	COMPLETE:				
		robot.release(sectionID);
		
		aoiLoad.material := '';
		aoiLoad.execute := FALSE;
		
		loadCornerCardboardsEx := TRUE;
END_CASE
END_METHOD

METHOD loadCornerGuards : BOOL
VAR_INPUT
	pairIndex : INT;
END_VAR
VAR_OUTPUT
	error : BOOL;
END_VAR
VAR
	pair : REFERENCE TO PositionMaterials REF= materialsArr[pairIndex];
	errorLeft, errorRight : BOOL;
END_VAR
{warning disable C0371}

loadCornerGuards := 
	loadCornerGuardsEx(
		robot:= robotLeft, 
		aoiLoad:= aoiCornerGuardLeft, 
		loadStep:= loadStepLeft, 
		pairIndex:= pairIndex, 
		includeTopLeft:= TRUE, 
		includeTopRight:= FALSE, 
		includeBottomLeft:= TRUE, 
		includeBottomRight:= FALSE, 
		error=> errorLeft) 
	AND
	loadCornerGuardsEx(
		robot:= robotRight, 
		aoiLoad:= aoiCornerGuardRight, 
		loadStep:= loadStepRight, 
		pairIndex:= pairIndex, 
		includeTopLeft:= FALSE, 
		includeTopRight:= TRUE, 
		includeBottomLeft:= FALSE, 
		includeBottomRight:= TRUE, 
		error=> errorRight);
		
error := errorLeft OR errorRight;

(*
IF robotLeft.error OR robotRight.error THEN
	error := TRUE;
	RETURN;
	
ELSIF 
	(robotLeft.reservation <> sectionID AND_THEN NOT robotLeft.reserve(sectionID)) OR 
	(robotRight.reservation <> sectionID AND_THEN NOT robotRight.reserve(sectionID))
THEN //loading requires both robots be reserved together
	RETURN;
	
ELSIF //robots have wrong tool
	(robotLeft.tool <> sectionID AND_THEN NOT robotLeft.changeEOAT(targetTool := sectionID)) OR
	(robotRight.tool <> sectionID AND_THEN NOT robotRight.changeEOAT(targetTool := sectionID))
THEN
	RETURN;
	
END_IF

CASE loadStep OF
	0: //top and bottom
		IF aoiCornerGuardLeft.done AND aoiCornerGuardRight.done THEN
			aoiCornerGuardLeft.execute := aoiCornerGuardRight.execute := FALSE;
			aoiCornerGuardLeft.material := aoiCornerGuardRight.material := '';
			loadStep := 10;
			RETURN;
		END_IF
		
		aoiCornerGuardLeft.suctions := 0;
		aoiCornerGuardLeft.surfaceID := Surface.TOP;
		aoiCornerGuardLeft.material := pair.top;
		aoiCornerGuardLeft.numPads := 0;
		
		aoiCornerGuardRight.suctions := suctionBottom;
		aoiCornerGuardRight.surfaceID := Surface.BOTTOM;
		aoiCornerGuardRight.material := pair.bottom;
		aoiCornerGuardRight.numPads := 0;
		
		aoiCornerGuardLeft.execute := NOT aoiCornerGuardLeft.done AND NOT aoiCornerGuardLeft.busy;
		aoiCornerGuardRight.execute := NOT aoiCornerGuardRight.done AND NOT aoiCornerGuardRight.busy;
		
	10: //sides
		IF aoiCornerGuardLeft.done AND aoiCornerGuardRight.done THEN
			aoiCornerGuardLeft.execute := aoiCornerGuardRight.execute := FALSE;
			aoiCornerGuardLeft.material := aoiCornerGuardRight.material := '';
			loadStep := 10;
			RETURN;
		END_IF
		
		aoiCornerGuardLeft.suctions := 0;
		aoiCornerGuardLeft.surfaceID := Surface.LEFT;
		aoiCornerGuardLeft.material := pair.left;
		aoiCornerGuardLeft.numPads := 0;
		
		aoiCornerGuardRight.suctions := 0;
		aoiCornerGuardRight.surfaceID := Surface.RIGHT;
		aoiCornerGuardRight.material := pair.right;
		aoiCornerGuardRight.numPads := 0;
		
		aoiCornerGuardLeft.execute := NOT aoiCornerGuardLeft.done AND NOT aoiCornerGuardLeft.busy;
		aoiCornerGuardRight.execute := NOT aoiCornerGuardRight.done AND NOT aoiCornerGuardRight.busy;
		
	COMPLETE:
		loadStep := 0;
		loadCornerGuards := TRUE;
END_CASE

error := aoiCornerGuardLeft.error OR aoiCornerGuardRight.error;
*)
END_METHOD

METHOD loadCornerGuardsEx : BOOL
VAR_IN_OUT
	robot : RobotA22;
	aoiLoad : AOI_LoadCornerGuard;
	loadStep : INT;
END_VAR
VAR_INPUT
	pairIndex : INT;
	includeTopLeft, includeTopRight, includeBottomLeft, includeBottomRight : BOOL;
END_VAR
VAR_OUTPUT
	error : BOOL;
END_VAR
VAR
	pair : REFERENCE TO PositionMaterials REF= materialsArr[pairIndex];
END_VAR
{warning disable C0371}
IF robot.error THEN
	error := TRUE;
	RETURN;
ELSIF robot.reservation <> sectionID AND_THEN NOT robot.reserve(sectionID) THEN
	RETURN;
ELSIF robot.tool <> sectionID AND_THEN NOT robot.changeEOAT(targetTool := sectionID) THEN
	RETURN;
END_IF

error := aoiLoad.error;

CASE loadStep OF
	0:
		loadStep := Surface.BOTTOM_LEFT;
		
	Surface.BOTTOM_LEFT:
		IF NOT includeBottomLeft OR aoiLoad.donePulse THEN
			aoiLoad.execute := FALSE;
			aoiLoad.material := '';
			loadStep := Surface.BOTTOM_RIGHT;
			RETURN;
		END_IF
		
		aoiLoad.surfaceID := loadStep;
		aoiLoad.material := pair.bottomLeft;
		aoiLoad.suctions := suctionBottomLeft;
		aoiLoad.numPads := UPPER_BOUND(suctionBottomLeft, 1) - LOWER_BOUND(suctionBottomLeft, 1) + 1;
		
		aoiLoad.execute := NOT aoiLoad.busy;
		
	Surface.BOTTOM_RIGHT:
		IF NOT includeBottomRight OR aoiLoad.donePulse THEN
			aoiLoad.execute := FALSE;
			aoiLoad.material := '';
			loadStep := Surface.TOP_LEFT;
			RETURN;
		END_IF
		
		aoiLoad.surfaceID := loadStep;
		aoiLoad.material := pair.bottomRight;
		aoiLoad.suctions := suctionBottomRight;
		aoiLoad.numPads := UPPER_BOUND(suctionBottomRight, 1) - LOWER_BOUND(suctionBottomRight, 1) + 1;
		
		aoiLoad.execute := NOT aoiLoad.busy;
	
	Surface.TOP_LEFT:		
		IF NOT includeTopLeft OR aoiLoad.donePulse THEN
			aoiLoad.execute := FALSE;
			aoiLoad.material := '';
			loadStep := Surface.TOP_RIGHT;
			RETURN;
		END_IF
		
		aoiLoad.surfaceID := loadStep;
		aoiLoad.material := pair.top;
		aoiLoad.suctions := suctionTopLeft;
		aoiLoad.numPads := UPPER_BOUND(suctionTopLeft, 1) - LOWER_BOUND(suctionTopLeft, 1) + 1;
		
		aoiLoad.execute := NOT aoiLoad.busy;
		
	Surface.TOP_RIGHT:
		IF NOT includeTopRight OR aoiLoad.donePulse THEN
			aoiLoad.execute := FALSE;
			aoiLoad.material := '';
			loadStep := COMPLETE;
			RETURN;
		END_IF
		
		aoiLoad.surfaceID := loadStep;
		aoiLoad.material := pair.topRight;
		aoiLoad.suctions := suctionTopRight;
		aoiLoad.numPads := UPPER_BOUND(suctionTopRight, 1) - LOWER_BOUND(suctionTopRight, 1) + 1;
		
		aoiLoad.execute := NOT aoiLoad.busy;
		
	COMPLETE:				
		robot.release(sectionID);
		
		aoiLoad.material := '';
		aoiLoad.execute := FALSE;
		
		loadCornerGuardsEx := TRUE;
END_CASE
END_METHOD

METHOD PROTECTED loadFlatCardboards : BOOL
VAR_INPUT
	pairIndex : INT;
END_VAR
VAR_OUTPUT
	error : BOOL;
END_VAR
VAR
	pair : REFERENCE TO PositionMaterials REF= materialsArr[pairIndex];
	errorLeft, errorRight : BOOL;
END_VAR
{warning disable C0371}

loadFlatCardboards := 
	loadFlatCardboardsEx(
		robot:= robotLeft, 
		aoiLoad:= aoiFlatCardboardLeft, 
		loadStep:= loadStepLeft, 
		pairIndex:= pairIndex, 
		includeTop:= TRUE, 
		includeLeft:= FALSE, //left already loaded before
		includeRight:= FALSE, 
		includeBottom:= FALSE, 
		error=> errorLeft)
	AND
	loadFlatCardboardsEx(
		robot:= robotRight, 
		aoiLoad:= aoiFlatCardboardRight, 
		loadStep:= loadStepRight, 
		pairIndex:= pairIndex, 
		includeTop:= FALSE, 
		includeLeft:= FALSE, 
		includeRight:= FALSE, //right already loaded before
		includeBottom:= TRUE, 
		error=> errorRight);
		
error := errorLeft OR errorRight;

(*
IF robotLeft.error OR robotRight.error THEN
	error := TRUE;
	RETURN;
	
ELSIF 
	(robotLeft.reservation <> sectionID AND_THEN NOT robotLeft.reserve(sectionID)) OR 
	(robotRight.reservation <> sectionID AND_THEN NOT robotRight.reserve(sectionID))
THEN //loading requires both robots be reserved together
	RETURN;
	
ELSIF //robots have wrong tool
	(robotLeft.tool <> sectionID AND_THEN NOT robotLeft.changeEOAT(targetTool := sectionID)) OR
	(robotRight.tool <> sectionID AND_THEN NOT robotRight.changeEOAT(targetTool := sectionID))
THEN
	RETURN;
	
END_IF

CASE loadStep OF
	0: //top and bottom
		IF aoiFlatCardboardLeft.done AND aoiFlatCardboardRight.done THEN
			aoiFlatCardboardLeft.execute := aoiFlatCardboardRight.execute := FALSE;
			aoiFlatCardboardLeft.material := aoiFlatCardboardRight.material := '';
			loadStep := 10;
			RETURN;
		END_IF
		
		aoiFlatCardboardLeft.suctions := 0;
		aoiFlatCardboardLeft.surfaceID := Surface.TOP;
		aoiFlatCardboardLeft.material := pair.top;
		aoiFlatCardboardLeft.numPads := 0;
		
		aoiFlatCardboardRight.suctions := suctionBottom;
		aoiFlatCardboardRight.surfaceID := Surface.BOTTOM;
		aoiFlatCardboardRight.material := pair.bottom;
		aoiFlatCardboardRight.numPads := 0;
		
		aoiFlatCardboardLeft.execute := NOT aoiFlatCardboardLeft.done AND NOT aoiFlatCardboardLeft.busy;
		aoiFlatCardboardRight.execute := NOT aoiFlatCardboardRight.done AND NOT aoiFlatCardboardRight.busy;
		
	10: //sides
		IF aoiFlatCardboardLeft.done AND aoiFlatCardboardRight.done THEN
			aoiFlatCardboardLeft.execute := aoiFlatCardboardRight.execute := FALSE;
			aoiFlatCardboardLeft.material := aoiFlatCardboardRight.material := '';
			loadStep := 10;
			RETURN;
		END_IF
		
		aoiFlatCardboardLeft.suctions := 0;
		aoiFlatCardboardLeft.surfaceID := Surface.LEFT;
		aoiFlatCardboardLeft.material := pair.left;
		aoiFlatCardboardLeft.numPads := 0;
		
		aoiFlatCardboardRight.suctions := 0;
		aoiFlatCardboardRight.surfaceID := Surface.RIGHT;
		aoiFlatCardboardRight.material := pair.right;
		aoiFlatCardboardRight.numPads := 0;
		
		aoiFlatCardboardLeft.execute := NOT aoiFlatCardboardLeft.done AND NOT aoiFlatCardboardLeft.busy;
		aoiFlatCardboardRight.execute := NOT aoiFlatCardboardRight.done AND NOT aoiFlatCardboardRight.busy;
		
	COMPLETE:
		loadStepLeft := loadStepRight := 0;
		loadStep := 0;
		
		loadFlatCardboards := TRUE;
END_CASE

error := aoiFlatCardboardLeft.error OR aoiFlatCardboardRight.error;
*)
END_METHOD

METHOD loadFlatCardboardsEx : BOOL
VAR_IN_OUT
	robot : RobotA22;
	aoiLoad : AOI_LoadFlatCardboard;
	loadStep : INT;
END_VAR
VAR_INPUT
	pairIndex : INT;
	includeTop, includeLeft, includeRight, includeBottom : BOOL;
END_VAR
VAR_OUTPUT
	error : BOOL;
END_VAR
VAR
	pair : REFERENCE TO PositionMaterials REF= materialsArr[pairIndex];
END_VAR
IF robot.error THEN
	error := TRUE;
	RETURN;
ELSIF robot.reservation <> sectionID AND_THEN NOT robot.reserve(sectionID) THEN
	RETURN;
ELSIF robot.tool <> sectionID AND_THEN NOT robot.changeEOAT(targetTool := sectionID) THEN
	RETURN;
END_IF

error := aoiLoad.error;

CASE loadStep OF
	0:
		loadStep := Surface.TOP;
	
	Surface.TOP:	
		IF NOT includeTop OR aoiLoad.donePulse THEN
			aoiLoad.execute := FALSE;
			aoiLoad.material := '';
			loadStep := Surface.BOTTOM;
			RETURN;
		END_IF
		
		aoiLoad.surfaceID := Surface.TOP;
		aoiLoad.material := pair.top;
		aoiLoad.suctions := 0;
		aoiLoad.numPads := 0;
		
		aoiLoad.execute := NOT aoiLoad.busy;
		
	Surface.BOTTOM:
		IF NOT includeBottom OR aoiLoad.donePulse THEN
			aoiLoad.execute := FALSE;
			aoiLoad.material := '';
			loadStep := Surface.LEFT;
			RETURN;
		END_IF
		
		aoiLoad.surfaceID := Surface.BOTTOM;
		aoiLoad.material := pair.bottom;
		aoiLoad.suctions := suctionBottom;
		aoiLoad.numPads := UPPER_BOUND(suctionBottom, 1) - LOWER_BOUND(suctionBottom, 1) + 1;
		
		aoiLoad.execute := NOT aoiLoad.busy;
		
	Surface.LEFT:
		IF NOT includeLeft OR aoiLoad.donePulse THEN
			aoiLoad.execute := FALSE;
			aoiLoad.material := '';
			loadStep := Surface.RIGHT;
			RETURN;
		END_IF
		
		aoiLoad.surfaceID := Surface.LEFT;
		aoiLoad.material := pair.left;
		aoiLoad.suctions := 0;
		aoiLoad.numPads := 0;
		
		aoiLoad.execute := NOT aoiLoad.busy;
		
	Surface.RIGHT:
		IF NOT includeRight OR aoiLoad.donePulse THEN
			aoiLoad.execute := FALSE;
			aoiLoad.material := '';
			loadStep := COMPLETE;
			RETURN;
		END_IF
		
		aoiLoad.surfaceID := Surface.RIGHT;
		aoiLoad.material := pair.right;
		aoiLoad.suctions := 0;
		aoiLoad.numPads := 0;
		
		aoiLoad.execute := NOT aoiLoad.busy;
		
	COMPLETE:				
		robot.release(sectionID);
		
		aoiLoad.material := '';
		aoiLoad.execute := FALSE;
		
		loadFlatCardboardsEx := TRUE;
END_CASE
END_METHOD

METHOD PROTECTED maintenance : BOOL
VAR_INPUT
END_VAR
{warning disable C0371}
IF robotLeft.Done THEN
	robotLeft.clearCommand();
END_IF

IF robotRight.Done THEN
	robotRight.clearCommand();
END_IF
END_METHOD

METHOD PROTECTED manual : BOOL
VAR_INPUT
END_VAR
END_METHOD

METHOD PROTECTED process : BOOL
VAR_INPUT
	auto : BOOL;
END_VAR
VAR_OUTPUT
	error : BOOL;
END_VAR
VAR
	currentPair : REFERENCE TO PositionMaterials REF= materialsArr[iPair];
END_VAR
{warning disable C0371}

IF iPair >= CONSTS.maxPairs THEN
	process := TRUE;
	RETURN;
ELSIF NOT PositionIsValid(pair := currentPair) THEN
	iPair := iPair + 1;
	RETURN;
END_IF
(*
corrected sequence:
	load sides
	load corners
	load bottom
	load top
*)

CASE step OF
	IDLE:
		IF execute THEN
			execute := FALSE;
			step := LOAD_SIDES_CORNERS;
		END_IF
	
	LOAD_SIDES_CORNERS:
		IF
			(auto AND done) OR
			(NOT auto AND execute)
		THEN
			aoiCornerCardboardLeft.reset();
			aoiCornerCardboardRight.reset();
			
			aoiCornerGuardLeft.reset();
			aoiCornerGuardRight.reset();
			
			aoiFlatCardboardLeft.reset();
			aoiFlatCardboardRight.reset();
			
			step := LOAD_TOP_BOTTOM;
			RETURN;
		END_IF
		
		IF NOT done THEN
			done := load(pairIndex := iPair);
		END_IF
		
	LOAD_TOP_BOTTOM:
		IF
			(auto AND done) OR
			(NOT auto AND execute)
		THEN
			aoiCornerCardboardLeft.reset();
			aoiCornerCardboardRight.reset();
			
			aoiCornerGuardLeft.reset();
			aoiCornerGuardRight.reset();
			
			aoiFlatCardboardLeft.reset();
			aoiFlatCardboardRight.reset();
			
			step := PUSH;
			RETURN;
		END_IF
		
		IF NOT done THEN
			done := loadFlatCardboards(pairIndex := iPair);
		END_IF
		
	PUSH:
		IF
			(auto AND latchLeft AND latchRight AND pistonBottom.extended) OR
			(NOT auto AND execute)
		THEN
			step := TARGET_WRAP_POSITION;
			RETURN;
		END_IF
		
		insertionLeft.align(demoHeight+5);
		insertionRight.align(demoHeight+5);
		
		IF //align slider to 5mm gap above bundle height
			insertionLeft.sliderPos <> demoHeight+5 OR
			insertionRight.sliderPos <> demoHeight+5
		THEN
			RETURN;
		END_IF
		
		IF NOT latchLeft THEN
			latchLeft := insertionLeft.contact;
			insertionLeft.press();
		END_IF
		
		IF NOT latchRight THEN
			latchRight := insertionRight.contact;
			insertionRight.press();
		END_IF
		
		pistonBottom.extend();
		
	TARGET_WRAP_POSITION:		
		IF iWrap >= wrapPoints THEN
			step := COMPLETE;
			RETURN;
		END_IF
		
		IF materialsArr[iPair].position = materialsArr[iPair + 1].position THEN //if this and the next pair were loaded together
			masterLength := TO_INT( MAX( GetPairMasterLength(materialsArr[iPair]), GetPairMasterLength(materialsArr[iPair + 1]) ) );
			wrapPoints := MAX( materialsArr[iPair].wrapPoints, materialsArr[iPair + 1].wrapPoints );
			wrapRotations := MAX( materialsArr[iPair].wrapRotations, materialsArr[iPair + 1].wrapRotations );
		ELSE
			masterLength := TO_INT( GetPairMasterLength(materialsArr[iPair]) );
			wrapPoints := materialsArr[iPair].wrapPoints;
			wrapRotations := materialsArr[iPair].wrapRotations;
		END_IF
		
		(*
		directionCheckAndSet(
			wrapConveyorPos,
			(currentPair.position - masterLength/2) + (masterLength/(currentPair.wrapPoints + 1) * (iWrap + 1)));
		*)
		step := WRAP_AND_RELEASE;
		
	WRAP_AND_RELEASE:
		releaseDelayTimer(IN:= , PT:= releaseDelay, Q=> , ET=> );
		
		IF wrapper.ready THEN
			wrapper.wrap(wrapRotations);
			releaseDelayTimer.IN := TRUE;
		END_IF
		
		IF releaseDelayTimer.Q THEN
			SetSuctions(suctions := suctionTopLeft, state := FALSE);
			SetSuctions(suctions := suctionTopRight, state := FALSE);
			SetSuctions(suctions := suctionBottomLeft, state := FALSE);
			SetSuctions(suctions := suctionBottomRight, state := FALSE);
			
			insertionLeft.toHome();
			insertionRight.toHome();
			pistonBottom.retract();
		END_IF
		
		IF wrapper.done AND insertionLeft.home AND insertionRight.home AND pistonBottom.retracted THEN
			releaseDelayTimer.IN := FALSE;
			step := WRAP_AND_RELEASE;
		END_IF
	
	COMPLETE:
		iPair := iPair + 1;
		iWrap := wrapPoints := wrapRotations := 0;
		step := IDLE;
		
END_CASE
END_METHOD

METHOD PROTECTED ps_AbortCondition : BOOL
VAR_INPUT
END_VAR
{warning disable C0371}
ps_AbortCondition :=
	insertionLeft.error OR 
	insertionRight.error OR 
	robotLeft.error OR 
	robotRight.error OR
	wrapper.error;
END_METHOD

METHOD PROTECTED ps_Aborted : BOOL
VAR_INPUT
END_VAR
ps_Aborted := TRUE;
END_METHOD

METHOD PROTECTED ps_Aborting : BOOL
VAR_INPUT
END_VAR
{warning disable C0371}
insertionLeft.stop();
insertionRight.stop();
pistonBottom.stop();

aoiFlatCardboardLeft.reset();
aoiFlatCardboardRight.reset();

aoiCornerCardboardLeft.reset();
aoiCornerCardboardRight.reset();

aoiCornerGuardLeft.reset();
aoiCornerGuardRight.reset();

robotLeft.clearCommand();
robotRight.clearCommand();

//stop conveyors

ps_Aborting :=
	NOT insertionLeft.active AND
	NOT insertionRight.active AND
	NOT pistonBottom.busy AND
	NOT robotLeft.Busy AND
	NOT robotRight.Busy;
END_METHOD

METHOD PROTECTED ps_Clearing : BOOL
VAR_INPUT
END_VAR
{warning disable C0371}
insertionLeft.reset();
insertionRight.reset();

ps_Clearing := 
	NOT insertionLeft.error AND
	NOT insertionRight.error AND
	NOT wrapper.error AND
	NOT robotLeft.error AND
	NOT robotRight.error;
END_METHOD

METHOD PROTECTED ps_Complete : BOOL
VAR_INPUT
END_VAR
ps_Complete := TRUE;
END_METHOD

METHOD PROTECTED ps_Completing : BOOL
VAR_INPUT
END_VAR
ps_Completing := NOT occupied;
END_METHOD

METHOD PROTECTED ps_Execute : BOOL
VAR_INPUT
END_VAR
VAR_OUTPUT
	error : BOOL;
END_VAR
CASE pmlMode OF
	0: //invalid mode
	ePMLCustomUnitMode_Production:		ps_Execute := process(auto := TRUE, error => error);
	ePMLCustomUnitMode_Maintenance:		ps_Execute := maintenance();
	ePMLCustomUnitMode_Manual:			ps_Execute := manual();
	ePMLCustomUnitMode_SemiAuto:		ps_Execute := process(auto := FALSE, error => error);
END_CASE
END_METHOD

METHOD PROTECTED ps_Held : BOOL
VAR_INPUT
END_VAR
ps_Held := NOT hold;
END_METHOD

METHOD PROTECTED ps_HoldCondition : BOOL
VAR_INPUT
END_VAR
END_METHOD

METHOD PROTECTED ps_Holding : BOOL
VAR_INPUT
END_VAR
{warning disable C0371}
insertionLeft.stop();
insertionRight.stop();
pistonBottom.stop();
//set robot to pause

ps_Holding :=
	NOT insertionLeft.active AND
	NOT insertionRight.active;
END_METHOD

METHOD PROTECTED ps_Idle : BOOL
VAR_INPUT
END_VAR
ps_Idle := execute;
execute := FALSE;
END_METHOD

METHOD PROTECTED ps_Resetting : BOOL
VAR_INPUT
END_VAR
{warning disable C0371}
insertionLeft.reset();
insertionRight.reset();

ps_Resetting := 
	reset AND
	NOT insertionLeft.error AND
	NOT insertionRight.error AND
	NOT wrapper.error AND
	NOT robotLeft.error AND
	NOT robotRight.error;
END_METHOD

METHOD PROTECTED ps_Starting : BOOL
VAR_INPUT
END_VAR
{warning disable C0371}
robotLeft.clearCommand();
robotRight.clearCommand();

insertionLeft.homingSequence();
insertionRight.homingSequence();
pistonBottom.retract();

ps_Starting := 
	insertionLeft.screw.HomeSet AND 
	insertionRight.screw.HomeSet AND 
	pistonBottom.retracted;
END_METHOD

METHOD PROTECTED ps_StopCondition : BOOL
VAR_INPUT
END_VAR
ps_StopCondition := 
	stop;
END_METHOD

METHOD PROTECTED ps_Stopped : BOOL
VAR_INPUT
END_VAR
ps_Stopped := TRUE;
END_METHOD

METHOD PROTECTED ps_Stopping : BOOL
VAR_INPUT
END_VAR
{warning disable C0371}
insertionLeft.stop();
insertionRight.stop();
pistonBottom.stop();

aoiFlatCardboardLeft.reset();
aoiFlatCardboardRight.reset();

aoiCornerCardboardLeft.reset();
aoiCornerCardboardRight.reset();

aoiCornerGuardLeft.reset();
aoiCornerGuardRight.reset();

robotLeft.clearCommand();
robotRight.clearCommand();

wrapper.bEnable := FALSE;

//stop conveyors

ps_Stopping :=
	//NOT insertionLeft.active AND
	NOT insertionRight.active AND
	NOT pistonBottom.busy AND
	NOT robotLeft.Busy AND
	NOT robotRight.Busy AND
	NOT wrapper.busy;
END_METHOD

METHOD PROTECTED ps_SuspendCondition : BOOL
VAR_INPUT
END_VAR
END_METHOD

METHOD PROTECTED ps_Suspended : BOOL
VAR_INPUT
END_VAR
ps_Suspended := NOT ps_SuspendCondition();
END_METHOD

METHOD PROTECTED ps_Suspending : BOOL
VAR_INPUT
END_VAR
ps_Suspending := TRUE;
END_METHOD

METHOD PROTECTED ps_Unholding : BOOL
VAR_INPUT
END_VAR
ps_Unholding := TRUE;
END_METHOD

METHOD PROTECTED ps_Unsuspending : BOOL
VAR_INPUT
END_VAR
ps_Unsuspending := TRUE;
END_METHOD

METHOD PROTECTED FINAL runSectionTasks : BOOL
VAR_INPUT
	auto : BOOL;
END_VAR
VAR_OUTPUT
	error : BOOL;
END_VAR
SUPER^.runSectionTasks(auto := auto, error => error);

CASE status OF
	SectionTask.IDLE:
		RETURN;
	
	SectionTask.ALIGNING:
		IF NOT recipesCombined THEN
			combine(
				currentBundle.cardboard, 
				currentBundle.cornerGuard, 
				materialsArr, 
				currentBundle.cardboard_over_cornerGuard);
				
			recipesCombined := TRUE;
		END_IF
		
	SectionTask.ACTIVE:
		recipesCombined := FALSE;
		
	SectionTask.CLEARING:
		//
		
	SectionTask.COMPLETE:	
		//
		
	-100:
		RETURN;
		
END_CASE
END_METHOD

METHOD PROTECTED setOrder : BOOL
VAR_IN_OUT
	innerArray : ARRAY[*] OF PositionMaterials;
	outerArray : ARRAY[*] OF PositionMaterials;
	
	combined : ARRAY[*] OF PositionMaterials;
	
	i_inner : INT;
	i_outer : INT;
	i_combined : INT;
END_VAR
VAR	
	outerMaterialLength : LREAL;
	innerMaterialLength : LREAL;
END_VAR
//if inner material is in front of outer material, inner material goes first
IF innerArray[i_inner].position <= outerArray[i_outer].position THEN

	combined[i_combined] := innerArray[i_inner];
	i_inner := i_inner + 1; //check next cardboard during next iteration
	
	setOrder := TRUE;
	RETURN;
END_IF
	
outerMaterialLength := GetPairMasterLength(outerArray[i_outer]);
innerMaterialLength := GetPairMasterLength(innerArray[i_inner]);

//if current inner material is too close to current outer material, place inner material first
//compare inner materials' front with outer material's back
IF (innerArray[i_inner].position - innerMaterialLength/2) < (outerArray[i_outer].position + outerMaterialLength/2) THEN
	combined[i_combined] := innerArray[i_inner];
	i_inner := i_inner + 1;
ELSE //otherwise, outer material can go
	combined[i_combined] := outerArray[i_outer];
	i_outer := i_outer + 1;
END_IF

setOrder := TRUE;
END_METHOD

METHOD PROTECTED unload : BOOL
VAR_INPUT
END_VAR
END_METHOD

END_FUNCTION_BLOCK

// ---- Sections/Abstract/SectionEx.TcPOU
FUNCTION_BLOCK ABSTRACT SectionEx
VAR_INPUT
	enable : BOOL;
	sectionID : SectionEnum;
END_VAR
VAR_IN_OUT
	bundlesQueue : ARRAY[*] OF Bundle;
	bundlesBypass : ARRAY[*] OF BOOL; //if true, then bypass current bundle
	
	conveyorsArr : ARRAY[*] OF POINTER TO ConveyorSC;
	//in addition to the conveyos array, each section must receive references to the origial conveyors the array elements point to
END_VAR
VAR_OUTPUT
	bundleOut : Bundle; //assigned if there is a bundle to target
	bypass : BOOL; //assigned once the bundle head passes the section (status >= ACTIVE)
END_VAR
VAR_OUTPUT //PackML states + controls
	run : BOOL;
	stop : BOOL;
	execute : BOOL;
	hold : BOOL;
	reset : BOOL;
	
	ready : BOOL;
	busy : BOOL;
	done : BOOL;
	error : BOOL;
	
	pmlModeString : STRING;
	pmlStateString : STRING;
	
	pmlState : E_PMLState;
	pmlMode : E_PMLCustomUnitMode;
	
	iBundle : INT(0..Consts.maxQueue);
	iPair : INT(0..Consts.maxPairs);
END_VAR
VAR //PackML types
	pmlCommand : E_PMLCommand;
	pmlModeRequest : E_PMLCustomUnitMode := ePMLCustomUnitMode_Production;
	
	pmlStateMachine : PML_StateMachine;
	pmlModeManager : PML_UnitModeManager;
	pmlSemiAutoConfig : PML_UnitModeConfig;
END_VAR
VAR
	currentBundle : REFERENCE TO Bundle;
	currentBypass : REFERENCE TO BOOL;
	
	loaded : BOOL;
	loadedMaterials : ARRAY[Surface.TOP..Surface.BOTTOM_RIGHT] OF STRING;
	
	entryRefPos : (*REFERENCE TO*) REAL;
	exitRefPos : (*REFERENCE TO*) REAL;
	
	requestedConveyorMode : ConveyorMode;
	
	nextSection : POINTER TO SectionEx;
	prevSection : POINTER TO SectionEx;
	
	occupied : BOOL; //may need to move this to Hardware GVL since this is a sensor
	
	status : SectionTask; //section status
END_VAR
VAR_STAT CONSTANT
	INCLUSIVE : INT := 0;
	EXCLUSIVE : INT := 1;
	COMPLETE : INT := 1030;
	
	suctionReleaseDelay : TIME := T#1000MS;
END_VAR

currentBundle REF= bundlesQueue[iBundle];
currentBypass REF= bundlesBypass[iBundle];
bypass := currentBypass;

ready := status = 0;
busy := status > 0;
done := done;
error := error;

blocks();

configPmlModes();
runPmlStates();

METHOD PROTECTED blocks : BOOL
pmlModeManager(
	bExecute:= NOT pmlModeManager.bExecute, 
	eModeCommand:= pmlModeRequest, 
	eState:= pmlState, 
	eModeStatus=> pmlMode, 
	sModeStatus=> pmlModeString, 
	bDone=> , 
	bError=> , 
	nErrorId=> );

pmlStateMachine(
	eMode:= pmlMode, 
	eCommand:= pmlCommand, 
	stSubUnitInfoRef:= , 
	stOptions:= , 
	eState=> pmlState, 
	sState=> pmlStateString, 
	bError=> , 
	nErrorID=> );
END_METHOD

METHOD PROTECTED configPmlModes : BOOL
pmlSemiAutoConfig(
	eMode:= 4, 
	sName:= 'SemiAuto', 
	bDisableClearing:= FALSE, 
	bDisableStarting:= FALSE, 
	bDisableSuspended:= FALSE, 
	bDisableStopping:= FALSE, 
	bDisableAborting:= FALSE, 
	bDisableHolding:= FALSE, 
	bDisableHeld:= FALSE, 
	bDisableUnholding:= FALSE, 
	bDisableSuspending:= FALSE, 
	bDisableUnsuspending:= FALSE, 
	bDisableResetting:= FALSE, 
	bDisableIdle:= FALSE, 
	bDisableCompleting:= FALSE, 
	bDisableComplete:= FALSE, 
	bEnableUnitModeChangeStopped:= TRUE, 
	bEnableUnitModeChangeIdle:= TRUE, 
	bEnableUnitModeChangeSuspended:= FALSE, 
	bEnableUnitModeChangeExecute:= FALSE, 
	bEnableUnitModeChangeAborted:= TRUE, 
	bEnableUnitModeChangeHeld:= FALSE, 
	bEnableUnitModeChangeComplete:= FALSE, 
	bError=> , 
	nErrorId=> );
END_METHOD

METHOD connectTo : BOOL
VAR_INPUT
	connectedSection : POINTER TO SectionEx;
END_VAR
nextSection := connectedSection;

IF connectedSection <> 0 THEN
	connectedSection^.prevSection := THIS;
END_IF
END_METHOD

METHOD PROTECTED directionCheckAndSet : BOOL
VAR_INPUT
	conveyorRef : REAL;
	target : REAL;
END_VAR
//returns true conveyorRef is in range of target
IF InRange(conveyorRef - CONSTS.precisionTolerance, conveyorRef + CONSTS.precisionTolerance, target, EXCLUSIVE) THEN
	directionCheckAndSet := TRUE;
	
ELSIF conveyorRef > target THEN
	pConveyorMode := ConveyorMode.BACKWARD;
	
ELSIF conveyorRef < target THEN
	pConveyorMode := ConveyorMode.FORWARD;
	
END_IF
END_METHOD

METHOD PROTECTED ABSTRACT load : BOOL
VAR_INPUT
	pairIndex : INT;
END_VAR
VAR_OUTPUT
	error : BOOL;
END_VAR
(*
loading takes place while the section is NOT active
materials are loaded for the next incoming bundle, not the current bundle - may differ for each section
*)
END_METHOD

METHOD PROTECTED ABSTRACT maintenance : BOOL
VAR_INPUT
END_VAR
END_METHOD

METHOD PROTECTED ABSTRACT manual : BOOL
VAR_INPUT
END_VAR
END_METHOD

PROPERTY PROTECTED pConveyorMode : ConveyorMode
GET
pConveyorMode := requestedConveyorMode;
END_GET
SET
VAR
	i : DINT;
END_VAR
requestedConveyorMode := pConveyorMode;

FOR i:=LOWER_BOUND(conveyorsArr, 1) TO UPPER_BOUND(conveyorsArr, 1) BY 1 DO
	
	CASE status OF
		SectionTask.ALIGNING, -100:
			//all conveyors requested to same mode
			conveyorsArr[i]^.setRequest(requestedConveyorMode);
			
		SectionTask.ACTIVE, SectionTask.CLEARING:
			//once previous bundle catches up, the conveyor that bundle sits on must be linked to this section
			//a conveyor control module will handle linking
			
			IF conveyorsArr[i]^.IsOccupied THEN //follow this section's request
				conveyorsArr[i]^.setRequest(requestedConveyorMode);
				
			ELSE //catch up succeeding bundle (FOLLOW PREVIOUS SECTION)
				IF prevSection <> 0 THEN
					conveyorsArr[i]^.setRequest( prevSection^.pConveyorMode );
				END_IF
			END_IF
	END_CASE	
	
END_FOR
END_SET
END_PROPERTY

METHOD PROTECTED ABSTRACT process : BOOL
VAR_INPUT
	auto : BOOL;
END_VAR
VAR_OUTPUT
	error : BOOL;
END_VAR
(*
this method is implemented by each section according to their material packaging steps
*)
END_METHOD

METHOD PROTECTED ABSTRACT ps_AbortCondition : BOOL
VAR_INPUT
END_VAR
END_METHOD

METHOD PROTECTED ABSTRACT ps_Aborted : BOOL
VAR_INPUT
END_VAR
END_METHOD

METHOD PROTECTED ABSTRACT ps_Aborting : BOOL
VAR_INPUT
END_VAR
END_METHOD

METHOD PROTECTED ABSTRACT ps_Clearing : BOOL
VAR_INPUT
END_VAR
END_METHOD

METHOD PROTECTED ABSTRACT ps_Complete : BOOL
VAR_INPUT
END_VAR
END_METHOD

METHOD PROTECTED ABSTRACT ps_Completing : BOOL
VAR_INPUT
END_VAR
END_METHOD

METHOD PROTECTED ps_Execute : BOOL
VAR_INPUT
END_VAR
VAR_OUTPUT
	error : BOOL;
END_VAR
CASE pmlMode OF
	0: //invalid mode
	ePMLCustomUnitMode_Production:		ps_Execute := runSectionTasks(auto := TRUE);
	ePMLCustomUnitMode_Maintenance:		ps_Execute := maintenance();
	ePMLCustomUnitMode_Manual:			ps_Execute := manual();
	ePMLCustomUnitMode_SemiAuto:		ps_Execute := runSectionTasks(auto := FALSE);
END_CASE
END_METHOD

METHOD PROTECTED ABSTRACT ps_Held : BOOL
VAR_INPUT
END_VAR
END_METHOD

METHOD PROTECTED ABSTRACT ps_HoldCondition : BOOL
VAR_INPUT
END_VAR
END_METHOD

METHOD PROTECTED ABSTRACT ps_Holding : BOOL
VAR_INPUT
END_VAR
END_METHOD

METHOD PROTECTED (*ABSTRACT*) ps_Idle : BOOL
VAR_INPUT
END_VAR
ps_Idle := run OR execute; (*start section input*)

IF execute THEN
	run := TRUE;
END_IF
END_METHOD

METHOD PROTECTED ABSTRACT ps_Resetting : BOOL
VAR_INPUT
END_VAR
END_METHOD

METHOD PROTECTED ABSTRACT ps_Starting : BOOL
VAR_INPUT
END_VAR
END_METHOD

METHOD PROTECTED ABSTRACT ps_StopCondition : BOOL
VAR_INPUT
END_VAR
END_METHOD

METHOD PROTECTED ABSTRACT ps_Stopped : BOOL
VAR_INPUT
END_VAR
END_METHOD

METHOD PROTECTED ABSTRACT ps_Stopping : BOOL
VAR_INPUT
END_VAR
END_METHOD

METHOD PROTECTED ABSTRACT ps_SuspendCondition : BOOL
VAR_INPUT
END_VAR
END_METHOD

METHOD PROTECTED ABSTRACT ps_Suspended : BOOL
VAR_INPUT
END_VAR
END_METHOD

METHOD PROTECTED ABSTRACT ps_Suspending : BOOL
VAR_INPUT
END_VAR
END_METHOD

METHOD PROTECTED ABSTRACT ps_Unholding : BOOL
VAR_INPUT
END_VAR
END_METHOD

METHOD PROTECTED ABSTRACT ps_Unsuspending : BOOL
VAR_INPUT
END_VAR
END_METHOD

PROPERTY PROTECTED pStatus : SectionTask
GET
pStatus := status;
END_GET
SET
status := pStatus;
END_SET
END_PROPERTY

METHOD PROTECTED runPmlStates : BOOL
(*
PackML
	state machine for packaging applications - see Tc3_PackML_V2 library on InfoSys
	
	final states - wait for an input or condition and command to new state
	intermediate states - complete a task and call pmlStateMachine.M_StateComplete() to advance to next state
	
the following states currently use the same logic (albeit in different methods), implementation may change later
	ps_Stopping() and ps_Aborting()
	ps_Resetting() and ps_Clearing()
	
STOP - controlled stop **with intent to shutdown or vacate for extended time** induced by operator/HMI - otherwise use HOLD
ABORT - emergency stop due to machine errors


HOLD - minor local issues
SUSPEND - external issues

EXECUTE - major control logic
	different modes may require different tasks
	create methods as required for different modes, then call the correct method in ps_Completing()
	can be commanded to STOP, ABORT, HOLD, or SUSPEND at any point
COMPLETING - process complete, move product out of system and finish transition to COMPLETED

the implementation below can be copied to all POUs that use a PackML state machine
the individual ps_< > methods need to be implemented for the specific application
*)


IF ps_AbortCondition() THEN //abort condition
	pmlCommand := ePMLCommand_Abort;
ELSIF ps_StopCondition() THEN //stop condition
	pmlCommand := ePMLCommand_Stop;
END_IF

CASE pmlState OF
	0 (*ePMLState_Undefined*): //default state on startup
		pmlCommand := ePMLCommand_Stop;
		
	ePMLState_Stopping:
		IF ps_Stopping() THEN
			pmlStateMachine.M_StateComplete();
		END_IF
		
	ePMLState_Stopped:
		IF ps_Stopped() THEN
			pmlCommand := ePMLCommand_Reset;
		END_IF
	
    ePMLState_Resetting:
		IF ps_Resetting() THEN
			pmlStateMachine.M_StateComplete();
		END_IF
		
	ePMLState_Idle:
		IF ps_Idle() THEN
			pmlCommand := ePMLCommand_Start;
		END_IF		
	
	ePMLState_Starting:
		IF ps_Starting() THEN
			pmlStateMachine.M_StateComplete();
		END_IF
	
	ePMLState_Execute: //check the conditions in order of their priority, currently HOLD has the highest priority
		IF ps_HoldCondition() THEN
			pmlCommand := ePMLCommand_Hold;
			
		ELSIF ps_SuspendCondition() THEN
			pmlCommand := ePMLCommand_Suspend;			
		
		ELSIF ps_Execute(error => error) THEN //ps_Execute.error => THIS^.error
			pmlStateMachine.M_StateComplete();
			pmlCommand := ePMLCommand_Complete;
		END_IF
		
	ePMLState_Completing:
		IF ps_Completing() THEN
			pmlStateMachine.M_StateComplete();
		END_IF
	
	ePMLState_Complete:
		IF ps_Complete() THEN
			pmlCommand := ePMLCommand_Reset;
		END_IF
	
	ePMLState_Holding:
		IF ps_Holding() THEN
			pmlStateMachine.M_StateComplete();
		END_IF
	
	ePMLState_Held:
		IF NOT hold THEN
			pmlCommand := ePMLCommand_Unhold;
		END_IF
	
	ePMLState_Unholding:
		IF ps_Unholding() THEN
			pmlStateMachine.M_StateComplete(); //release all pause commands and IO
		END_IF
		
	ePMLState_Suspending: //based on next section conditions
		IF ps_Suspending() THEN
			pmlStateMachine.M_StateComplete();
		END_IF
		
	ePMLState_Suspended: //based on next section conditions
		IF ps_Suspended() THEN
			pmlCommand := ePMLCommand_Unsuspend;
		END_IF
	
	ePMLState_Unsuspending: //based on next section conditions
		IF ps_Unsuspending() THEN
			pmlStateMachine.M_StateComplete();
		END_IF
	
	ePMLState_Aborting:
		IF ps_Aborting() THEN
			pmlStateMachine.M_StateComplete();
		END_IF
	
	ePMLState_Aborted:
		IF ps_Aborted() THEN
			pmlCommand := ePMLCommand_Clear;
		END_IF
	
	ePMLState_Clearing:
		IF ps_Clearing() THEN
			pmlStateMachine.M_StateComplete();
		END_IF
	
END_CASE
END_METHOD

METHOD PROTECTED runSectionTasks : BOOL
VAR_INPUT
	auto : BOOL;
END_VAR
VAR_OUTPUT
	error : BOOL;
END_VAR
CASE status OF
	SectionTask.IDLE:
		IF BundleIsValid(currentBundle) THEN			
			status := SectionTask.ALIGNING;
			done := FALSE;
		END_IF
	
	SectionTask.ALIGNING:		
		pConveyorMode := ConveyorMode.FORWARD;
		
		IF 
			occupied AND
			nextSection <> 0 AND
			nextSection^.pConveyorMode = ConveyorMode.BACKWARD
		THEN //section occupied by next section backing up into this section
			status := -100;
			
		ELSIF occupied THEN //section occupied by correct bundle
			//stop and zero the conveyors
			IF NOT auto OR_ELSE execute THEN
				status := SectionTask.ACTIVE;
			END_IF
		END_IF
		
	SectionTask.ACTIVE:
		bundleOut := currentBundle;
		
		IF NOT enable THEN
			iPair := 0;
			status := SectionTask.CLEARING;
			
		ELSIF currentBypass (*AND_THEN discharge()*) THEN //bundle failed in previous section, discharge this section's materials
			IF unload() THEN
				iPair := 0;
				status := SectionTask.CLEARING;
			END_IF
			
		ELSIF process(auto := auto, error => error) THEN //bundle recipe completed normally
			IF NOT auto OR_ELSE execute THEN
				iPair := 0;
				status := SectionTask.CLEARING;
			END_IF			
		END_IF
		
	SectionTask.CLEARING:
		bundleOut := currentBundle;
		pConveyorMode := ConveyorMode.FORWARD;
		
		IF exitRefPos >= currentBundle.length AND NOT occupied THEN //rear of bundle has cleared the area
			status := SectionTask.COMPLETE;
		END_IF
		
	SectionTask.COMPLETE:	
		iBundle := iBundle + 1;
		//bundleOut := GVL.nullBundle;
		MEMSET(ADR(bundleOut), 0, SIZEOF(bundleOut));
		
		status := SectionTask.IDLE;
		
		runSectionTasks := TRUE;
		
	-100: //previously completed bundle reversed into this section		
		pConveyorMode := ConveyorMode.FORWARD;
		
		IF NOT occupied THEN
			status := SectionTask.ALIGNING;
		END_IF
		
END_CASE
END_METHOD

METHOD shiftIterator : BOOL
//2023-10-24 - array of pointers replaced with iterator for MAIN's queue passed by pointer
iBundle := iBundle - 1;
END_METHOD

METHOD PROTECTED ABSTRACT unload : BOOL
VAR_INPUT
END_VAR
(*
unload, unstage, etc
*)
END_METHOD

END_FUNCTION_BLOCK

// ---- Sections/A22 - Cardboard/AOIs/AOI_LoadCornerGuard.TcPOU
FUNCTION_BLOCK AOI_LoadCornerGuard
VAR_INPUT
	execute : BOOL;
END_VAR
VAR_IN_OUT CONSTANT
	sectionID : SectionEnum;
END_VAR
VAR_IN_OUT
	robot : RobotA22;
	magazine : SkidMagazine;
	loadedMaterials : ARRAY[*] OF STRING;
END_VAR
VAR_INPUT
	surfaceID : Surface;
	material : STRING;
	
	suctions : POINTER TO SuctionPad; //access from 0 to numPads-1, not LOWER_BOUND to UPPER_BOUND
	numPads : DINT;
END_VAR
VAR_OUTPUT
	donePulse : BOOL; //this signal turns on 1 cycle after done turns true, should not affect the program structure
	done : BOOL;
	busy : BOOL;
	error : BOOL;
	
	recovery : BOOL;
	failCounter : INT;
END_VAR
VAR
	run : BOOL;
	trigger : R_TRIG;
	doneTrigger : R_TRIG;
	
	column : INT;
	
	suctionTimer : TON;
	step : (IDLE, PREP_ROBOT, GET_FROM_STORAGE, LOAD_TO_INSERTION, COMPLETE, RECOVERY_IDLE, RECOVERY_REMOVE, RECOVERY_LOAD);
	
	i : DINT;
END_VAR
VAR CONSTANT
	suctionDelay : TIME := T#2S;
	suctionDistance : INT := 10;
END_VAR

{warning disable C0371}

trigger(CLK:= execute, Q=> );
doneTrigger(CLK:= done, Q=> donePulse);
busy := trigger.Q OR step > 0;

IF step > IDLE AND_THEN NOT preExecution() THEN //conditions to track before execution
	RETURN;
END_IF

(*
if required bunk was not found on table - restage entire table
if bunk was not loaded correctly - remove bunk, then restage entire table
*)
CASE step OF
	IDLE:
		IF trigger.Q THEN
			recovery := FALSE;
			done := FALSE;
			error := FALSE;
			step := PREP_ROBOT;
		END_IF
		
	PREP_ROBOT:
		robot.clearCommand();
		IF robot.Ready THEN
			step := GET_FROM_STORAGE;
			column := 0;
		END_IF
		
	GET_FROM_STORAGE:		
		IF NOT magazine.findSlot(material := material, index => column) THEN
			error := TRUE;
			RETURN;
		END_IF
		
		IF robot.eoatDistance < suctionDistance THEN //move from table to robot gripper
			robot.HoldMaterial := magazine.getSlot(i := column, error => );
		END_IF
		
		IF robot.Done THEN
			step := COMPLETE;
			RETURN;
		ELSIF robot.materialAtHoldingPosition > 0 THEN
			step := LOAD_TO_INSERTION;
			RETURN;
		END_IF
		
		CASE surfaceID OF
			Surface.TOP_LEFT, Surface.TOP_RIGHT:			robot.setGroup(group := 1, value := TaskA22.LOAD_CORNER_GUARD_UPPER);
			Surface.BOTTOM_LEFT, SURFACE.BOTTOM_RIGHT:		robot.setGroup(group := 1, value := TaskA22.LOAD_CORNER_GUARD_LOWER);
		END_CASE
		robot.setGroup(group := 2, value := column); 
			
	LOAD_TO_INSERTION:
		IF robot.materialAtHoldingPosition > 0 AND robot.HoldMaterial <> '' THEN //move from gripper to insertion
			loadedMaterials[surfaceID] := robot.HoldMaterial;
			robot.HoldMaterial := '';
		END_IF
		
		//numPads/3 <= i < numPads/3 * 2
		FOR i:=(numPads/3)*1 TO (numPads/3)*2-1 BY 1 DO //middle third suctions only
			suctions[i].enable := TRUE;
		END_FOR
		
		IF robot.Done THEN
			suctionTimer.IN := FALSE;
			step := COMPLETE;
			RETURN;
		END_IF
		
		suctionTimer(IN:= , PT:= suctionDelay, Q=> , ET=> );
		suctionTimer.IN := TRUE;
		
		IF suctionTimer.Q THEN
			robot.setGroup(group := 10, value := robot.materialAtHoldingPosition);
		END_IF
	
	COMPLETE:
		robot.clearCommand();
		
		IF //check insertion quality
			SuctionQualityPtr(
				suctions := suctions, 
				numPads := numPads, 
				insertionMaterial := loadedMaterials[surfaceID], 
				recipeMaterial := material)
		THEN
			done := TRUE;
			column := 0;
			step := 0;
			
		ELSE //recovery - remove and reload
			failCounter := failCounter + 1;
			step := RECOVERY_IDLE;
		END_IF
		
	//---------RECOVERY-----------------------------------------
	RECOVERY_IDLE:
		robot.clearCommand();
		IF robot.Ready THEN
			step := RECOVERY_REMOVE;
		END_IF
		
	RECOVERY_REMOVE:
		IF robot.Done THEN
			step := RECOVERY_LOAD;
			RETURN;
		END_IF
		
		CASE surfaceID OF
			Surface.TOP_LEFT, Surface.TOP_RIGHT:			robot.setGroup(group := 1, value := TaskA22.REMOVE_CORNER_GUARD_UPPER);
			Surface.BOTTOM_LEFT, SURFACE.BOTTOM_RIGHT:		robot.setGroup(group := 1, value := TaskA22.REMOVE_CORNER_GUARD_LOWER);
		END_CASE
		
	RECOVERY_LOAD:	
		recovery := TRUE;
		error := TRUE;
		
END_CASE

METHOD PRIVATE preExecution : BOOL
VAR_INPUT
END_VAR
{warning disable C0371}
IF material = '' THEN
	done := TRUE;
	RETURN;
END_IF

IF //robot must be ready before execution
	robot.error OR 
	robot.reservation <> sectionID OR 
	robot.tool <> sectionID
THEN
	error := TRUE;
	RETURN;
END_IF

preExecution := TRUE;
END_METHOD

METHOD reset : BOOL
VAR_INPUT
END_VAR
done := FALSE;
busy := FALSE;
error := FALSE;
recovery := FALSE;
failCounter := 0;

column := 0;
step := 0;
END_METHOD

END_FUNCTION_BLOCK

// ---- Sections/A22 - Cardboard/AOIs/AOI_LoadCornerCardboard.TcPOU
FUNCTION_BLOCK AOI_LoadCornerCardboard
VAR_INPUT
	execute : BOOL;
END_VAR
VAR_IN_OUT CONSTANT
	sectionID : SectionEnum;
END_VAR
VAR_IN_OUT
	robot : RobotA22;
	skid : SkidMagazine;
	loadedMaterials : ARRAY[*] OF STRING;
	overheadTray : STRING;
END_VAR
VAR_INPUT
	surfaceID : Surface;
	material : STRING;
	
	suctions : POINTER TO SuctionPad; //access from 0 to numPads-1, not LOWER_BOUND to UPPER_BOUND
	numPads : DINT;
	
	hasBendingMachine : BOOL;
	foldPos0 : INT;
	foldPos1 : INT;
END_VAR
VAR_OUTPUT
	donePulse : BOOL; //this signal turns on 1 cycle after done turns true and remains on for 1 cycle
	done : BOOL;
	busy : BOOL;
	error : BOOL;
	
	recovery : BOOL;
	failCounter : INT;
END_VAR
VAR
	run : BOOL;
	trigger : R_TRIG;
	doneTrigger : R_TRIG;
	
	column : INT;
	
	suctionTimer : TON;
	
	step : (IDLE, PREP_ROBOT, //common
			GET_FROM_STORAGE, PLACE_TO_OVERHEAD, //left robot only
			GET_FROM_OVERHEAD, //right robot only
			LOAD_TO_INSERTION, COMPLETE, RECOVERY_IDLE, RECOVERY_REMOVE, RECOVERY_LOAD); //common
	
	i : DINT;
END_VAR
VAR CONSTANT
	suctionDelay : TIME := T#2S;
	suctionDistance : INT := 10;
END_VAR

{warning disable C0371}

trigger(CLK:= execute, Q=> );
doneTrigger(CLK:= done, Q=> donePulse);
busy := trigger.Q OR step > 0;

IF step > IDLE AND_THEN NOT preExecution() THEN //conditions to track before execution
	RETURN;
END_IF

CASE step OF
	IDLE:
		IF trigger.Q THEN
			step := PREP_ROBOT;
		END_IF
		
	PREP_ROBOT:
		robot.clearCommand();
		IF robot.Ready THEN
			IF NOT hasBendingMachine THEN //IMPORTANT - this condition differentiates left and right sequences
				step := GET_FROM_STORAGE;
			ELSE
				step := GET_FROM_OVERHEAD;
			END_IF
		END_IF
		
	//----------LEFT ROBOT----------------------------------------
	GET_FROM_STORAGE:
		_GetFromStorage();
	
	PLACE_TO_OVERHEAD:
		_PlaceToOverhead();
	
	//----------RIGHT ROBOT----------------------------------------
	GET_FROM_OVERHEAD:
		_GetFromOverhead();
		
	//----------COMMON----------------------------------------
	LOAD_TO_INSERTION:
		_LoadToInsertion();
		
	COMPLETE:
		robot.clearCommand();

		IF //check insertion quality
			SuctionQualityPtr(
				suctions := suctions,
				numPads := numPads, 
				insertionMaterial := loadedMaterials[surfaceID], 
				recipeMaterial := material) 
		THEN
			done := TRUE;
			column := 0;
			step := 0;
			
		ELSE //recovery
			failCounter := failCounter + 1;
			step := RECOVERY_IDLE;
		END_IF
		
	RECOVERY_IDLE:
		robot.clearCommand();
		IF robot.Ready THEN
			step := RECOVERY_REMOVE;
		END_IF
		
	RECOVERY_REMOVE:
		IF robot.Done THEN
			step := RECOVERY_LOAD;
			RETURN;
		END_IF
	
		CASE surfaceID OF
			Surface.TOP_RIGHT:		robot.setGroup(group := 1, value := TaskA22.REMOVE_CARDBOARD_UPPER_CORNER);
			Surface.BOTTOM_RIGHT:	robot.setGroup(group := 1, value := TaskA22.REMOVE_CARDBOARD_LOWER_CORNER);
		END_CASE
		
	RECOVERY_LOAD:
		error := TRUE;
		recovery := TRUE;
			
		IF hasBendingMachine THEN
			step := 0;
		END_IF
		
END_CASE

METHOD PRIVATE _Complete : BOOL
VAR_INPUT
END_VAR
{warning disable C0371}
robot.clearCommand();

IF //check insertion quality
	SuctionQualityPtr(
		suctions := suctions,
		numPads := numPads, 
		insertionMaterial := loadedMaterials[surfaceID], 
		recipeMaterial := material) 
THEN
	done := TRUE;
	column := 0;
	step := 0;
	
ELSE //recovery
	failCounter := failCounter + 1;
	step := RECOVERY_IDLE;
END_IF
END_METHOD

METHOD PRIVATE _GetFromOverhead : BOOL
VAR_INPUT
END_VAR
{warning disable C0371}
IF overheadTray = '' AND robot.HoldMaterial = '' THEN
	RETURN;
END_IF

IF robot.eoatDistance < suctionDistance THEN
	robot.HoldMaterial := overheadTray;
	overheadTray := '';
END_IF

IF robot.Done THEN
	step := COMPLETE;
	RETURN;
ELSIF robot.materialAtHoldingPosition > 0 THEN
	step := LOAD_TO_INSERTION;
	RETURN;
END_IF

CASE surfaceID OF
	Surface.TOP_RIGHT:		robot.setGroup(group := 1, value := TaskA22.LOAD_OVERHEAD_TO_UPPER_CORNER);
	Surface.BOTTOM_RIGHT:	robot.setGroup(group := 1, value := TaskA22.LOAD_OVERHEAD_TO_LOWER_CORNER);
END_CASE
robot.setGroup(group := 2, value := 0);
robot.setGroup(group := 3, value := 0);
END_METHOD

METHOD PRIVATE _GetFromStorage : BOOL
VAR_INPUT
END_VAR
{warning disable C0371}
IF NOT skid.findSlot(material := material, index=> column) THEN
	error := TRUE;
	RETURN;
END_IF

IF robot.eoatDistance < suctionDistance THEN
	robot.HoldMaterial := skid.getSlot(i := column);
END_IF

IF robot.Done THEN
	
	CASE surfaceID OF //determine what to do with the cardboard - load to insertion or move to overhead tray
		Surface.TOP_RIGHT, Surface.BOTTOM_RIGHT:	step := PLACE_TO_OVERHEAD;
		Surface.TOP_LEFT, Surface.BOTTOM_LEFT:		step := LOAD_TO_INSERTION;
	END_CASE
	
	RETURN;
END_IF

robot.setGroup(group := 1, value := TaskA22.TRANSFER_TO_BENDER);
robot.setGroup(group := 2, value := foldPos0);
robot.setGroup(group := 3, value := foldPos1);
END_METHOD

METHOD PRIVATE _LoadToInsertion : BOOL
VAR_INPUT
END_VAR
{warning disable C0371}
FOR i:=(numPads/3)*0 TO (numPads/3)*1 - 1 BY 1 DO //first third suctions only
	suctions[i].enable := TRUE;
END_FOR

FOR i:=(numPads/3)*2 TO (numPads/3)*3 - 1 BY 1 DO //last third suctions only
	suctions[i].enable := TRUE;
END_FOR

IF robot.Done THEN
	suctionTimer.IN := FALSE;
	step := COMPLETE;
	RETURN;
END_IF

suctionTimer(IN:= , PT:= suctionDelay, Q=> , ET=> );
suctionTimer.IN := TRUE;

IF suctionTimer.Q THEN
	robot.setGroup(group := 10, value := robot.materialAtHoldingPosition);
END_IF
END_METHOD

METHOD PRIVATE _PlaceToOverhead : BOOL
VAR_INPUT
END_VAR
{warning disable C0371}
IF robot.Done THEN
	step := COMPLETE;
	RETURN;
END_IF

robot.setGroup(group := 1, value := TaskA22.TRANSFER_TO_OVERHEAD);
robot.setGroup(group := 2, value := 0);
robot.setGroup(group := 3, value := 0);
END_METHOD

METHOD PRIVATE preExecution : BOOL
VAR_INPUT
END_VAR
{warning disable C0371}
IF material = '' THEN
	done := TRUE;
	RETURN;
END_IF

IF //robot must be ready before execution
	robot.error OR 
	robot.reservation <> sectionID OR 
	robot.tool <> sectionID
THEN
	error := TRUE;
	RETURN;
END_IF

preExecution := TRUE;
END_METHOD

METHOD reset : BOOL
VAR_INPUT
END_VAR
done := FALSE;
busy := FALSE;
error := FALSE;
recovery := FALSE;
failCounter := 0;

column := 0;
step := 0;
END_METHOD

END_FUNCTION_BLOCK

// ---- Sections/A22 - Cardboard/AOIs/AOI_LoadFlatCardboard.TcPOU
FUNCTION_BLOCK AOI_LoadFlatCardboard
VAR_INPUT
	execute : BOOL;
END_VAR
VAR_IN_OUT CONSTANT
	sectionID : SectionEnum;
END_VAR
VAR_IN_OUT
	robot : RobotA22;
	skid : SkidMagazine;
	loadedMaterials : ARRAY[*] OF STRING;
END_VAR
VAR_INPUT
	surfaceID : Surface;
	material : STRING;
	
	suctions : POINTER TO SuctionPad; //access from 0 to numPads-1, not LOWER_BOUND to UPPER_BOUND
	numPads : DINT;
END_VAR
VAR_OUTPUT
	donePulse : BOOL;
	done : BOOL;
	busy : BOOL;
	error : BOOL;
	
	recovery : BOOL;
	failCounter : INT;
END_VAR
VAR
	run : BOOL;
	trigger : R_TRIG;
	doneTrigger : R_TRIG;
	
	column : INT;
	
	suctionTimer : TON;
	step : (IDLE, PREP_ROBOT, GET_FROM_STORAGE, LOAD_TO_INSERTION, COMPLETE, RECOVERY_IDLE, RECOVERY_REMOVE, RECOVERY_WAIT, RECOVERY_LOAD);
	
	i : DINT;
END_VAR
VAR_STAT CONSTANT
	suctionDelay : TIME := T#2S;
	suctionDistance : INT := 10;
END_VAR

{warning disable C0371}

trigger(CLK:= execute, Q=> );
doneTrigger(CLK:= done, Q=> donePulse);
busy := trigger.Q OR step > 0;

IF step > IDLE AND_THEN NOT preExecution() THEN //conditions to track before execution
	RETURN;
END_IF

(*
if bunk was not loaded correctly - remove bunk, then restage entire table
*)
CASE step OF
	IDLE:
		IF trigger.Q THEN
			recovery := FALSE;
			done := FALSE;
			error := FALSE;
			step := PREP_ROBOT;
		END_IF
		
	PREP_ROBOT:
		robot.clearCommand();
		IF robot.Ready THEN
			step := GET_FROM_STORAGE;
			column := 0;
		END_IF
		
	GET_FROM_STORAGE:		
		IF NOT skid.findSlot(material := material, index => column) THEN
			error := TRUE;
			RETURN;
		END_IF
		
		IF robot.eoatDistance < suctionDistance THEN//move from table to robot gripper
			robot.HoldMaterial := skid.getSlot(i := column, error => );;
		END_IF
		
		IF robot.Done THEN
			step := COMPLETE;
			RETURN;
		ELSIF robot.materialAtHoldingPosition >= 1 AND robot.materialAtHoldingPosition <= 8 THEN
			step := LOAD_TO_INSERTION;
			RETURN;
		END_IF
		
		CASE surfaceID OF
			Surface.TOP_LEFT, Surface.TOP_RIGHT:			robot.setGroup(group := 1, value := TaskA22.LOAD_CORNER_GUARD_UPPER);
			Surface.BOTTOM_LEFT, SURFACE.BOTTOM_RIGHT:		robot.setGroup(group := 1, value := TaskA22.LOAD_CORNER_GUARD_LOWER);
		END_CASE
		robot.setGroup(group := 2, value := column); 
			
	LOAD_TO_INSERTION:
		IF robot.materialAtHoldingPosition > 0 AND robot.HoldMaterial <> '' THEN //move from gripper to insertion
			loadedMaterials[surfaceID] := robot.HoldMaterial;
			robot.HoldMaterial := '';
		END_IF
		
		//only bottom cardboard uses suction
		CASE surfaceID OF
			Surface.BOTTOM:		SetSuctionsPtr(suctions := suctions, numPads := numPads, state := TRUE);
		END_CASE
		
		IF robot.Done THEN
			suctionTimer.IN := FALSE;
			step := COMPLETE;
			RETURN;
		END_IF
		
		suctionTimer(IN:= , PT:= suctionDelay, Q=> , ET=> );
		suctionTimer.IN := TRUE;
		
		IF suctionTimer.Q THEN
			robot.setGroup(group := 10, value := robot.materialAtHoldingPosition);
		END_IF
	
	COMPLETE:
		robot.clearCommand();
		
		IF //if bottom then check insertion, otherwise done
			surfaceID <> Surface.BOTTOM OR_ELSE 
			SuctionQualityPtr(
				suctions := suctions, 
				numPads := numPads, 
				insertionMaterial := loadedMaterials[surfaceID], 
				recipeMaterial := material)
		THEN
			done := TRUE;
			column := 0;
			step := 0;
			
		ELSE //recovery - remove and reload
			failCounter := failCounter + 1;
			step := RECOVERY_IDLE;
		END_IF
		
	//---------RECOVERY-----------------------------------------
	RECOVERY_IDLE:
		robot.clearCommand();
		IF robot.Ready THEN
			step := RECOVERY_REMOVE;
		END_IF
		
	RECOVERY_REMOVE:
		IF robot.Done THEN
			step := RECOVERY_LOAD;
			RETURN;
		END_IF
		
		CASE surfaceID OF
			Surface.BOTTOM:		robot.setGroup(group := 1, value := TaskA22.REMOVE_CARDBOARD_BOTTOM);
		END_CASE
		
	RECOVERY_LOAD:	
		recovery := TRUE;
		error := TRUE;
		
END_CASE

METHOD PRIVATE preExecution : BOOL
VAR_INPUT
END_VAR
{warning disable C0371}
IF material = '' THEN
	done := TRUE;
	RETURN;
END_IF

IF //robot must be ready before execution
	robot.error OR 
	robot.reservation <> sectionID OR 
	robot.tool <> sectionID
THEN
	error := TRUE;
	RETURN;
END_IF

preExecution := TRUE;
END_METHOD

METHOD reset : BOOL
VAR_INPUT
END_VAR
done := FALSE;
busy := FALSE;
error := FALSE;
recovery := FALSE;
failCounter := 0;

column := 0;
step := 0;
END_METHOD

END_FUNCTION_BLOCK

// ---- Sections/A21a - Chipboard/ChipboardEx.TcPOU
FUNCTION_BLOCK ChipboardEx EXTENDS SectionEx
VAR_IN_OUT
	A21_SC_C18 : ConveyorSC;
	A21_LSC_C19 : ConveyorLSC;
	A21_LSC_C20 : ConveyorLSC;
END_VAR
VAR_IN_OUT
	robotLeft, robotRight : RobotA21;
	toolStorageLeft, toolStorageRight : A21ToolStorage;
	
	skidLeft, skidRight : SkidMagazine;
END_VAR
VAR	
	step : (IDLE, RETRACT_CONVEYOR, LOAD_CIP, EXTEND_CONVEYOR, COMPLETE := 1050);
	
	loadSet : INT;
END_VAR
VAR //bundle data
	materialsArr : (*REFERENCE TO*) ARRAY[0..Consts.maxPairs] OF PositionMaterials;
END_VAR
VAR
	aoiLoadLeft, aoiLoadRight : AOI_LoadChipboard;
	
	pushSmallConveyorPos : REAL;
	pushLargeConveyorPos : REAL;
END_VAR

aoiBlocks(); //call AOIs and large library FBs

SUPER^();

METHOD PROTECTED aoiBlocks : BOOL
VAR_INPUT
END_VAR
{warning disable C0371}
aoiLoadRight(
	sectionID:= sectionID, 
	execute:= ,
	robot:= robotRight, 
	storage:= skidRight,
	loadedMaterials:= loadedMaterials,
	surfaceID:= , 
	material:= , 
	loadedMaterials=> , 
	done=> , 
	error=> );
	
aoiLoadRight(
	sectionID:= sectionID, 
	execute:= , 
	robot:= robotRight, 
	storage:= skidRight,
	loadedMaterials:= loadedMaterials, 
	surfaceID:= , 
	material:= , 
	busy=> , 
	done=> , 
	error=> , 
	recovery=> , 
	failCounter=> );
END_METHOD

METHOD PROTECTED load : BOOL
VAR_INPUT
	pairIndex : INT;
END_VAR
VAR_OUTPUT
	error : BOOL;
END_VAR
VAR
	pair : REFERENCE TO PositionMaterials REF= materialsArr[pairIndex];
END_VAR
{warning disable C0371}
IF robotLeft.error AND robotLeft.error THEN
	error := TRUE;
	RETURN;

ELSIF
	( robotLeft.reservation <> sectionID AND_THEN robotLeft.reserve(sectionID) ) OR
	( robotRight.reservation <> sectionID AND_THEN robotRight.reserve(sectionID) ) THEN
	RETURN;
	
ELSIF //wrong tool and not finished changing tool
	(robotLeft.tool <> sectionID AND_THEN NOT robotLeft.changeEOAT(targetTool := sectionID)) OR
	(robotRight.tool <> sectionID AND_THEN NOT robotRight.changeEOAT(targetTool := sectionID))
THEN
	RETURN;
END_IF
//robots ok

CASE loadSet OF
	0: //left robot -> top, right robot -> bottom
		IF aoiLoadLeft.done AND aoiLoadRight.done THEN
			aoiLoadLeft.execute := aoiLoadRight.execute := FALSE;
			loadSet := 10;
			RETURN;
		END_IF
		
		aoiLoadLeft.surfaceID := Surface.TOP;
		aoiLoadLeft.material := pair.left;
		
		aoiLoadRight.surfaceID := Surface.BOTTOM;
		aoiLoadRight.material := pair.right;
		
		aoiLoadLeft.execute := NOT aoiLoadLeft.recovery;
		aoiLoadRight.execute := NOT aoiLoadRight.recovery;
		
	10: //recovery		
		IF robotRight.error THEN //left ok, right error
			
			IF aoiLoadLeft.done THEN
				aoiLoadLeft.execute := FALSE;
				loadSet := COMPLETE;
				RETURN;
			END_IF
			
			aoiLoadLeft.surfaceID := Surface.BOTTOM;
			aoiLoadLeft.material := pair.bottom;
			aoiLoadLeft.execute := NOT aoiLoadLeft.recovery;
			
		ELSIF robotLeft.error THEN //left error, right ok
			
			IF aoiLoadRight.done THEN
				aoiLoadRight.execute := FALSE;
				loadSet := COMPLETE;
				RETURN;
			END_IF
			
			aoiLoadRight.surfaceID := Surface.TOP;
			aoiLoadRight.material := pair.top;
			aoiLoadRight.execute := NOT aoiLoadRight.recovery;
			
		END_IF
		
	COMPLETE:
		loadSet := 0;
		
		robotLeft.release(sectionID);
		robotRight.release(sectionID);
		
		load := TRUE;
END_CASE
END_METHOD

METHOD PRIVATE loadingSequence : BOOL
VAR_IN_OUT
	robot : RobotA21;
	storage : SkidMagazine;
	loadStep : INT;
END_VAR
VAR_INPUT
	surfaceID : Surface;
	material : STRING;
END_VAR
VAR_OUTPUT
	fail : BOOL;
END_VAR
VAR
	slot : INT;
END_VAR
VAR CONSTANT
	suctionDistance : INT := 10;
END_VAR
{warning disable C0371}
IF material = '' THEN
	loadingSequence := TRUE;
	RETURN;
END_IF

CASE loadStep OF
	0:
		robot.clearCommand();
		IF robot.Ready THEN
			loadStep := 1;
		END_IF
	
	1:
		IF surfaceID = Surface.BOTTOM (*AND_THEN conveyors not retracted*) THEN
			//retract conveyors
			RETURN;
		END_IF
		loadStep := 10;
		
	10: //grab from chipboard skid
		IF NOT storage.findSlot(material := material, index => slot) THEN
			fail := TRUE;
			RETURN;
		(*
		ELSIF surfaceID = Surface.BOTTOM (*AND_THEN (*conveyor not lowered*)*) THEN
			//lower conveyor
			RETURN;
		*)
		END_IF
		
		IF robot.eoatDistance < suctionDistance THEN
			robot.HoldMaterial := storage.getSlot(i := slot);
		END_IF
		
		IF robot.Done THEN
			loadStep := COMPLETE;
			RETURN;
		ELSIF robot.materialAtHoldingPosition.4 OR robot.materialAtHoldingPosition.5 THEN //bits 4 and 5 are chipboard in position
			loadStep := 20;
			RETURN;
		END_IF
		
		robot.setGroup(group := 1, value := TaskA21.PLACE_CHIPBOARD_TOP);
		robot.setGroup(group := 2, value := slot);
		
	20: //place to bundle
		IF robotLeft.Done THEN
			loadStep := COMPLETE;
			RETURN;
		END_IF
		
		IF robot.HoldMaterial <> '' THEN
			loadedMaterials[surfaceID] := robot.HoldMaterial;
			robot.HoldMaterial := '';
		END_IF
		
	COMPLETE:
		IF loadedMaterials[surfaceID] = material THEN
			loadingSequence := TRUE;
		ELSE
			loadStep := 0;
		END_IF
		
END_CASE
END_METHOD

METHOD PROTECTED maintenance : BOOL
VAR_INPUT
END_VAR
{warning disable C0371}
//no specific tasks yet, free run and testing

IF robotLeft.Done THEN
	robotLeft.clearCommand();
END_IF

IF robotRight.Done THEN
	robotRight.clearCommand();
END_IF
END_METHOD

METHOD PROTECTED manual : BOOL
VAR_INPUT
END_VAR
END_METHOD

METHOD PROTECTED process : BOOL
VAR_INPUT
	auto : BOOL;
END_VAR
VAR_OUTPUT
	error : BOOL;
END_VAR
CASE step OF
	IDLE:
		IF execute THEN
			execute := FALSE;
			step := RETRACT_CONVEYOR;
		END_IF
		
	RETRACT_CONVEYOR:
		(*
		IF demoPair.bottom <> '' (*retract conveyors*) THEN
			IF TRUE (*BLSC 1-3 retracted*) THEN
				done := TRUE;
			END_IF
		ELSE
			done := TRUE;
		END_IF
		
		IF
			(manualStep AND_THEN execute) OR
			(NOT manualStep AND_THEN done)
		THEN
			done := FALSE;
			step := LOAD_MATERIAL;
		END_IF
		*)
		step := LOAD_CIP;
	LOAD_CIP:
		IF NOT done THEN
			done := load(pairIndex:= iPair, error=> error);
		END_IF
		
		IF
			(auto AND done) OR
			(NOT auto AND_THEN execute)
		THEN
			done := FALSE;
			execute := FALSE;
			
			step := EXTEND_CONVEYOR;
		END_IF
		
	EXTEND_CONVEYOR:
		(*
		IF FALSE (*conveyors not extended*) THEN
			//extend conveyors
		END_IF
		
		IF
			(auto AND done) OR
			(NOT auto AND_THEN execute) //conveyors extended
		THEN
			done := FALSE;
			step := COMPLETE;
		END_IF
		*)
		step := COMPLETE;
	COMPLETE:
		//reset everything
		step := IDLE;
		
		process := TRUE;
		
END_CASE
END_METHOD

METHOD PROTECTED ps_AbortCondition : BOOL
VAR_INPUT
END_VAR
{warning disable C0371}
ps_AbortCondition :=
	robotLeft.error OR 
	robotRight.error;
END_METHOD

METHOD PROTECTED ps_Aborted : BOOL
VAR_INPUT
END_VAR
ps_Aborted := TRUE;
END_METHOD

METHOD PROTECTED ps_Aborting : BOOL
VAR_INPUT
END_VAR
{warning disable C0371}
aoiLoadLeft.reset();
aoiLoadRight.reset();

robotLeft.clearCommand();
robotRight.clearCommand();

//stop conveyors

ps_Aborting :=
	NOT robotLeft.Busy AND
	NOT robotRight.Busy;
END_METHOD

METHOD PROTECTED ps_Clearing : BOOL
VAR_INPUT
END_VAR
{warning disable C0371}
(*reset conveyors*)

ps_Clearing := 
	NOT robotLeft.error AND
	NOT robotRight.error;
END_METHOD

METHOD PROTECTED ps_Complete : BOOL
VAR_INPUT
END_VAR
ps_Complete := TRUE;
END_METHOD

METHOD PROTECTED ps_Completing : BOOL
VAR_INPUT
END_VAR
ps_Completing := NOT occupied;
END_METHOD

METHOD PROTECTED ps_Execute : BOOL
VAR_INPUT
END_VAR
VAR_OUTPUT
	error : BOOL;
END_VAR
CASE pmlMode OF
	0: //invalid mode
	ePMLCustomUnitMode_Production:	ps_Execute := process(auto := FALSE, error => error);
	ePMLCustomUnitMode_Maintenance:	maintenance();
	ePMLCustomUnitMode_Manual:		ps_Execute := process(auto := TRUE, error => error);
END_CASE
END_METHOD

METHOD PROTECTED ps_Held : BOOL
VAR_INPUT
END_VAR
ps_Held := NOT hold;
END_METHOD

METHOD PROTECTED ps_HoldCondition : BOOL
VAR_INPUT
END_VAR
END_METHOD

METHOD PROTECTED ps_Holding : BOOL
VAR_INPUT
END_VAR
{warning disable C0371}
//set robot to pause

ps_Holding := TRUE;
END_METHOD

METHOD PROTECTED ps_Idle : BOOL
VAR_INPUT
END_VAR
ps_Idle := execute;
execute := FALSE;
END_METHOD

METHOD PROTECTED ps_Resetting : BOOL
VAR_INPUT
END_VAR
{warning disable C0371}
(*reset conveyors*)

ps_Resetting := 
	reset AND
	NOT robotLeft.error AND
	NOT robotRight.error;
END_METHOD

METHOD PROTECTED ps_Starting : BOOL
VAR_INPUT
END_VAR
{warning disable C0371}
//extend conveyors

ps_Starting := TRUE; //conveyors extended
END_METHOD

METHOD PROTECTED ps_StopCondition : BOOL
VAR_INPUT
END_VAR
ps_StopCondition := 
	stop;
END_METHOD

METHOD PROTECTED ps_Stopped : BOOL
VAR_INPUT
END_VAR
ps_Stopped := TRUE;
END_METHOD

METHOD PROTECTED ps_Stopping : BOOL
VAR_INPUT
END_VAR
{warning disable C0371}
aoiLoadLeft.reset();
aoiLoadRight.reset();

robotLeft.clearCommand();
robotRight.clearCommand();

//stop conveyors

ps_Stopping :=
	NOT robotLeft.Busy AND
	NOT robotRight.Busy;
END_METHOD

METHOD PROTECTED ps_SuspendCondition : BOOL
VAR_INPUT
END_VAR
END_METHOD

METHOD PROTECTED ps_Suspended : BOOL
VAR_INPUT
END_VAR
ps_Suspended := NOT ps_SuspendCondition();
END_METHOD

METHOD PROTECTED ps_Suspending : BOOL
VAR_INPUT
END_VAR
ps_Suspending := TRUE;
END_METHOD

METHOD PROTECTED ps_Unholding : BOOL
VAR_INPUT
END_VAR
ps_Unholding := TRUE;
END_METHOD

METHOD PROTECTED ps_Unsuspending : BOOL
VAR_INPUT
END_VAR
ps_Unsuspending := TRUE;
END_METHOD

METHOD PROTECTED runSectionTasks : BOOL
VAR_INPUT
	auto : BOOL;
END_VAR
VAR_OUTPUT
	error : BOOL;
END_VAR
SUPER^.runSectionTasks(auto := auto, error => error);

CASE status OF //add additional instructions for each state
	SectionTask.IDLE:
		//
	
	SectionTask.ALIGNING:
		//
		
	SectionTask.ACTIVE:
		//
		
	SectionTask.CLEARING:
		aoiLoadLeft.reset();
		aoiLoadRight.reset();
		
	SectionTask.COMPLETE:	
		//
		
	-100:
		RETURN;
		
END_CASE
END_METHOD

METHOD PROTECTED unload : BOOL
VAR_INPUT
END_VAR
//unload from insertion
//remove from staging table
END_METHOD

END_FUNCTION_BLOCK

// ---- Sections/A21a - Chipboard/AOIs/AOI_LoadChipboard.TcPOU
FUNCTION_BLOCK AOI_LoadChipboard
VAR_IN_OUT CONSTANT
	sectionID : SectionEnum;
END_VAR
VAR_INPUT
	execute : BOOL;
END_VAR
VAR_IN_OUT
	robot : RobotA21;
	storage : SkidMagazine;
	loadedMaterials : ARRAY[*] OF STRING;
END_VAR
VAR_INPUT
	surfaceID : Surface;
	material : STRING;
END_VAR
VAR_OUTPUT
	busy : BOOL;
	done : BOOL;
	error : BOOL;
	
	recovery : BOOL;
	failCounter : INT;
	
	donePulse : BOOL;
END_VAR
VAR
	run : BOOL;
	trigger : R_TRIG;
	doneTrigger : R_TRIG;
	
	step : (IDLE, PREP_ROBOT, RETRACT_CONVEYORS, GET_FROM_SKID, LOAD_TO_BUNDLE, COMPLETE);
	column : INT;
END_VAR
VAR CONSTANT
	suctionDistance : INT := 10;
END_VAR

{warning disable C0371}

trigger(CLK:= execute, Q=> );
doneTrigger(CLK:= done, Q=> donePulse);
busy := trigger.Q OR step > 0;

IF step > IDLE AND_THEN NOT preExecution() THEN //conditions to track before execution
	RETURN;
END_IF

trigger(CLK:= execute, Q=> run);

CASE step OF
	IDLE:
		IF trigger.Q THEN //reset outputs
			done := FALSE;
			error := FALSE;
			recovery := FALSE;
			
			step := PREP_ROBOT;
		END_IF
	
	PREP_ROBOT:
		robot.clearCommand();
		IF robot.Ready THEN
			step := RETRACT_CONVEYORS;
		END_IF
	
	RETRACT_CONVEYORS:
		IF surfaceID = Surface.BOTTOM (*AND_THEN conveyors not retracted*) THEN
			//retract conveyors
			RETURN;
		END_IF
		step := GET_FROM_SKID;
		
	GET_FROM_SKID: //grab from chipboard skid
		IF NOT storage.findSlot(material := material, index => column) THEN
			error := TRUE;
			RETURN;
		(*
		ELSIF surfaceID = Surface.BOTTOM (*AND_THEN (*conveyor not lowered*)*) THEN
			//lower conveyor
			RETURN;
		*)
		END_IF
		
		IF robot.eoatDistance < suctionDistance THEN
			robot.HoldMaterial := storage.getSlot(i := column);
		END_IF
		
		IF robot.Done THEN
			step := COMPLETE;
			RETURN;
		ELSIF robot.materialAtHoldingPosition.4 OR robot.materialAtHoldingPosition.5 THEN //bits 4 and 5 = chipboard in position
			step := LOAD_TO_BUNDLE;
			RETURN;
		END_IF
		CASE surfaceID OF
			Surface.TOP:		robot.setGroup(group := 1, value := TaskA21.PLACE_CHIPBOARD_TOP);
			Surface.BOTTOM:		robot.setGroup(group := 1, value := TaskA21.PLACE_CHIPBOARD_BOTTOM);
		END_CASE
		robot.setGroup(group := 2, value := column);
		
	LOAD_TO_BUNDLE: //place to bundle
		IF robot.Done THEN
			step := COMPLETE;
			RETURN;
		END_IF
		
		IF robot.HoldMaterial <> '' THEN
			loadedMaterials[surfaceID] := robot.HoldMaterial;
			robot.HoldMaterial := '';
		END_IF
		
	COMPLETE:
		IF loadedMaterials[surfaceID] = material THEN
			done := TRUE;
			failCounter := 0;
		ELSE
			error := TRUE;
			failCounter := failCounter + 1;
		END_IF
		step := 0;
END_CASE

busy := run OR step > 0;

METHOD PRIVATE preExecution : BOOL
VAR_INPUT
END_VAR
{warning disable C0371}
IF material = '' THEN
	done := TRUE;
	RETURN;
END_IF

IF //robot must be ready before execution
	robot.error OR 
	robot.reservation <> sectionID OR 
	robot.tool <> sectionID
THEN
	error := TRUE;
	RETURN;
END_IF

preExecution := TRUE;
END_METHOD

METHOD reset : BOOL
VAR_INPUT
END_VAR
VAR
	temp : AOI_LoadChipboard;
END_VAR
//(*
done := FALSE;
error := FALSE;
recovery := FALSE;
column := 0;
step := 0;

failCounter := 0;
//*)
//THIS^ := temp;
END_METHOD

END_FUNCTION_BLOCK

// ---- Sections/A21b - Wood Bunk/WoodBunkEx.TcPOU
FUNCTION_BLOCK WoodBunkEx EXTENDS SectionEx
VAR_IN_OUT
	A21_LSC_C21 : ConveyorLSC;
END_VAR
VAR_IN_OUT
	robotLeft, robotRight : RobotA21;
	toolStorageLeft, toolStorageRight : A21ToolStorage;
	
	stagingTableLeft, stagingTableRight : StagingTable;
	magazineLeft, magazineRight : SkidMagazine;
	
	strapper : StrapMachine;
	
	insertionLeft, insertionRight : Insertion;
	pistonBottom : SimplePiston;
	
	suctionTop : ARRAY[*] OF SuctionPad; (*1..3*)
	suctionLeft : ARRAY[*] OF SuctionPad; (*1..4*)
	suctionRight : ARRAY[*] OF SuctionPad; (*1..4*)
	suctionBottom : ARRAY[*] OF SuctionPad; (*1..2*)
END_VAR
VAR
	conveyorPos : REAL; //may need to move this to SectionEx
	
	step : (IDLE, STAGING, LOAD_WB, PUSH, STRAP, RELEASE, COMPLETE := 1050);
	
	stageStepLeft, stageStepRight : INT;
	loadStepLeft, loadStepRight : INT;
END_VAR
VAR //bundle data
	demoHeight : REAL := 640; //mm
	materialsArr : (*REFERENCE TO*) ARRAY[0..CONSTS.maxPairs] OF PositionMaterials;
END_VAR
VAR
	//AOIs encapsulate functionality and reduce the number of module variables
	aoiTemplateLeft, aoiTemplateRight : AOI_StagingTemplate;
	aoiStageLeft, aoiStageRight : AOI_StageWoodBunk; 
	aoiLoadLeft, aoiLoadRight : AOI_LoadWoodBunk;
	
	suctionRelease : TON;
	
	//for testing, to be removed when deployoed
	latchLeft, latchRight : BOOL; //prevents SMC sliders from overshooting
	suctionEnableTop, suctionEnableLeft, suctionEnableRight, suctionEnableBottom : BOOL;
END_VAR

aoiBlocks();

SUPER^();

(*
any PackML state-methods that SectionEx has a concrete implementation for will be overriden by concrete FBs that extend it
(ie: all or most of them)

to call the base implementation, add:
	SUPER^.ps_<state>();
to the concrete FB's implementation of that state-method
*)

METHOD PROTECTED aoiBlocks : BOOL
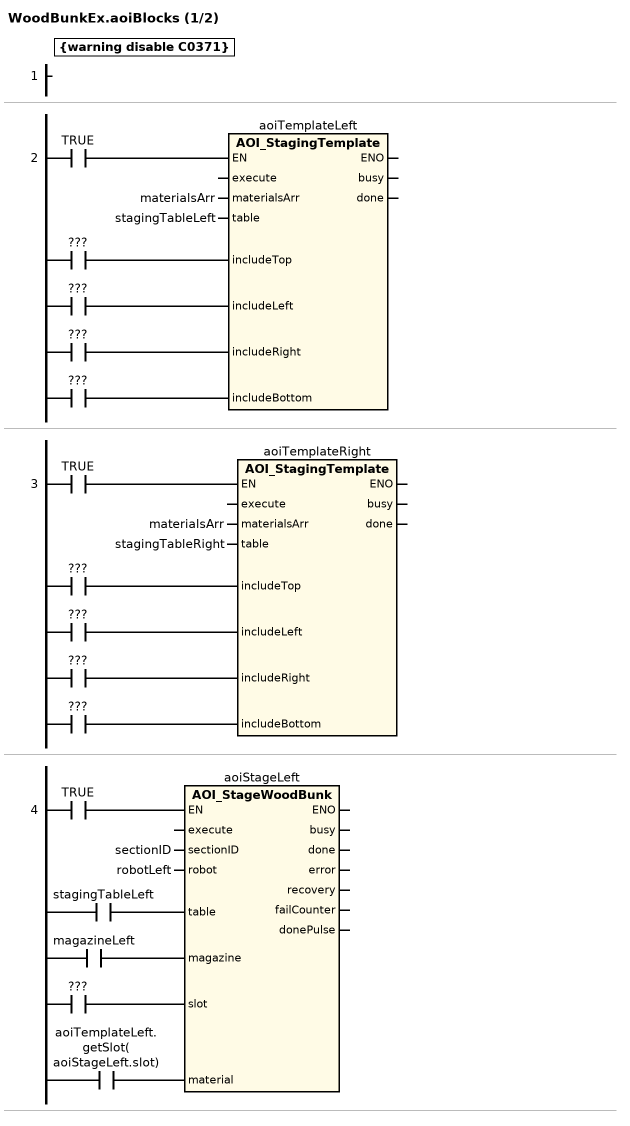
// NETWORK 1
// label: {warning disable C0371}

// NETWORK 2
aoiTemplateLeft(materialsArr := materialsArr, table := stagingTableLeft); // AOI_StagingTemplate

// NETWORK 3
aoiTemplateRight(materialsArr := materialsArr, table := stagingTableRight); // AOI_StagingTemplate

// NETWORK 4
aoiStageLeft(
    sectionID := sectionID,
    robot := robotLeft,
    table := stagingTableLeft,
    magazine := magazineLeft,
    material := aoiTemplateLeft.getSlot(aoiStageLeft.slot)); // AOI_StageWoodBunk

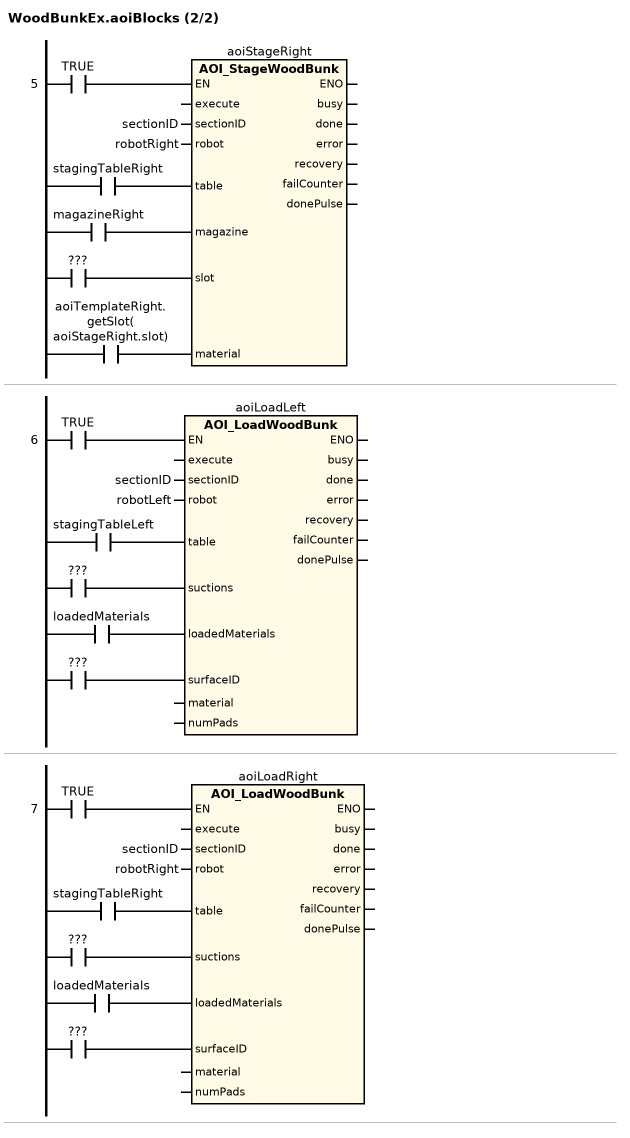
// NETWORK 5
aoiStageRight(
    sectionID := sectionID,
    robot := robotRight,
    table := stagingTableRight,
    magazine := magazineRight,
    material := aoiTemplateRight.getSlot(aoiStageRight.slot)); // AOI_StageWoodBunk

// NETWORK 6
aoiLoadLeft(
    sectionID := sectionID,
    robot := robotLeft,
    table := stagingTableLeft,
    loadedMaterials := loadedMaterials); // AOI_LoadWoodBunk

// NETWORK 7
aoiLoadRight(
    sectionID := sectionID,
    robot := robotRight,
    table := stagingTableRight,
    loadedMaterials := loadedMaterials); // AOI_LoadWoodBunk
END_METHOD

METHOD PROTECTED load : BOOL
VAR_INPUT
	pairIndex : INT;
END_VAR
VAR_OUTPUT
	error : BOOL;
END_VAR
VAR
	pair : REFERENCE TO PositionMaterials REF= materialsArr[pairIndex];
	errorLeft, errorRight : BOOL;
END_VAR
{warning disable C0371}
(*
this is the new code for loading wood bunks from staging table to insertion
loading sequences are independent as each side has its own step variable
can be extended by changing the include<> parameters
*)

load :=
	loadEx(
		robot:= robotLeft, 
		aoiLoad:= aoiLoadLeft, 
		loadStep:= loadStepLeft, 
		pairIndex:= pairIndex, 
		includeTop:= TRUE, 
		includeLeft:= TRUE, 
		includeRight:= FALSE, 
		includeBottom:= FALSE, 
		error=> errorLeft)
	AND
	loadEx(
		robot:= robotRight, 
		aoiLoad:= aoiLoadRight, 
		loadStep:= loadStepRight, 
		pairIndex:= pairIndex, 
		includeTop:= FALSE, 
		includeLeft:= FALSE, 
		includeRight:= TRUE, 
		includeBottom:= TRUE, 
		error=> errorRight);
		
error := errorLeft OR errorRight;

(*
below is the old code for loading wood bunks from staging table to insertion
it loads wood bunks in sets - top/bottom, then sides
if one side is finished loading a set before the other, it waits until the other side is done before advancing the set
*)
(*
IF robotLeft.error OR robotRight.error THEN
	error := TRUE;
	RETURN;
	
ELSIF 
	(robotLeft.reservation <> sectionID AND_THEN NOT robotLeft.reserve(sectionID)) OR 
	(robotRight.reservation <> sectionID AND_THEN NOT robotRight.reserve(sectionID))
THEN //loading requires both robots be reserved together
	RETURN;
	
ELSIF //robots have wrong tool
	(robotLeft.tool <> sectionID AND_THEN NOT robotLeft.changeEOAT(targetTool := sectionID)) OR
	(robotRight.tool <> sectionID AND_THEN NOT robotRight.changeEOAT(targetTool := sectionID))
THEN
	RETURN;
	
END_IF

CASE loadStep OF
	0: //top and bottom
		IF aoiLoadLeft.done AND aoiLoadRight.done THEN
			aoiLoadLeft.execute := aoiLoadRight.execute := FALSE;
			aoiLoadLeft.material := aoiLoadRight.material := '';
			
			aoiLoadLeft.reset();
			aoiLoadRight.reset();
			loadStep := 10;
			RETURN;
		END_IF
		
		aoiLoadLeft.suctions := suctionTop;
		aoiLoadLeft.surfaceID := Surface.TOP;
		aoiLoadLeft.material := pair.top;
		aoiLoadLeft.numPads := UPPER_BOUND(suctionTop, 1) - LOWER_BOUND(suctionTop, 1) + 1;
		
		aoiLoadRight.suctions := suctionBottom;
		aoiLoadRight.surfaceID := Surface.BOTTOM;
		aoiLoadRight.material := pair.bottom;
		aoiLoadRight.numPads := UPPER_BOUND(suctionBottom, 1) - LOWER_BOUND(suctionBottom, 1) + 1;
		
		aoiLoadLeft.execute := NOT aoiLoadLeft.done AND NOT aoiLoadLeft.busy;
		aoiLoadRight.execute := NOT aoiLoadRight.done AND NOT aoiLoadRight.busy;
		
	10: //sides
		IF aoiLoadLeft.done AND aoiLoadRight.done THEN
			aoiLoadLeft.execute := aoiLoadRight.execute := FALSE;
			aoiLoadLeft.material := aoiLoadRight.material := '';
			
			aoiLoadLeft.reset();
			aoiLoadRight.reset();
			loadStep := COMPLETE;
			RETURN;
		END_IF
		
		aoiLoadLeft.suctions := suctionLeft;
		aoiLoadLeft.surfaceID := Surface.LEFT;
		aoiLoadLeft.material := pair.left;
		aoiLoadLeft.numPads := UPPER_BOUND(suctionLeft, 1) - LOWER_BOUND(suctionLeft, 1) + 1;
		
		aoiLoadRight.suctions := suctionRight;
		aoiLoadRight.surfaceID := Surface.RIGHT;
		aoiLoadRight.material := pair.right;
		aoiLoadRight.numPads := UPPER_BOUND(suctionRight, 1) - LOWER_BOUND(suctionRight, 1) + 1;
		
		aoiLoadLeft.execute := NOT aoiLoadLeft.done AND NOT aoiLoadLeft.busy;
		aoiLoadRight.execute := NOT aoiLoadRight.done AND NOT aoiLoadRight.busy;
		
	COMPLETE:				
		robotLeft.release(sectionID);
		robotRight.release(sectionID);
		
		aoiLoadLeft.material := aoiLoadRight.material := '';
		aoiLoadLeft.execute := aoiLoadRight.execute := FALSE;
		
		loadStep := 0;
		load := TRUE;
END_CASE

//--------------------------------------------------
IF aoiLoadLeft.recovery THEN //if loading in recovery mode - refill table, resume loading when finished
	aoiLoadLeft.execute := stageEx(
		robot:= robotLeft, 
		aoiTemplate:= aoiTemplateLeft, 
		aoiStaging:= aoiStageLeft, 
		stageStep:= stageStepLeft, 
		includeTop:= TRUE, 
		includeLeft:= TRUE, 
		includeRight:= FALSE, 
		includeBottom:= FALSE, 
		error=> );
ELSE
	//loadLeft.execute := NOT loadLeft.busy AND NOT loadLeft.done;
END_IF
//--------------------------------------------------
IF aoiLoadRight.recovery THEN
	aoiLoadRight.execute := stageEx(
		robot:= robotRight, 
		aoiTemplate:= aoiTemplateRight, 
		aoiStaging:= aoiStageRight, 
		stageStep:= stageStepRight, 
		includeTop:= FALSE, 
		includeLeft:= FALSE, 
		includeRight:= TRUE, 
		includeBottom:= TRUE, 
		error=> );
ELSE
	//loadRight.execute := NOT loadRight.busy AND NOT loadRight.done;
END_IF
//--------------------------------------------------
	
error := aoiLoadLeft.error OR aoiLoadRight.error;
*)
END_METHOD

METHOD PRIVATE loadEx : BOOL
VAR_IN_OUT
	robot : RobotA21;
	aoiLoad : AOI_LoadWoodBunk;
	loadStep : INT;
END_VAR
VAR_INPUT
	pairIndex : INT;
	includeTop, includeLeft, includeRight, includeBottom : BOOL;
END_VAR
VAR_OUTPUT
	error : BOOL;
END_VAR
VAR
	pair : REFERENCE TO PositionMaterials REF= materialsArr[pairIndex];
END_VAR
{warning disable C0371}
IF robot.error THEN
	error := TRUE;
	RETURN;
ELSIF robot.reservation <> sectionID AND_THEN NOT robot.reserve(sectionID) THEN
	RETURN;
ELSIF robot.tool <> sectionID AND_THEN NOT robot.changeEOAT(targetTool := sectionID) THEN
	RETURN;
END_IF

error := aoiLoad.error;

CASE loadStep OF
	0:
		loadStep := Surface.TOP;
	
	Surface.TOP:		
		IF NOT includeTop OR aoiLoad.donePulse THEN
			aoiLoad.execute := FALSE;
			aoiLoad.material := '';
			loadStep := Surface.BOTTOM;
			RETURN;
		END_IF
		
		aoiLoad.surfaceID := Surface.TOP;
		aoiLoad.material := pair.top;
		aoiLoad.suctions := suctionTop;
		aoiLoad.numPads := UPPER_BOUND(suctionTop, 1) - LOWER_BOUND(suctionTop, 1) + 1;
		
		aoiLoad.execute := NOT aoiLoad.busy;
		
	Surface.BOTTOM:
		IF NOT includeBottom OR aoiLoad.donePulse THEN
			aoiLoad.execute := FALSE;
			aoiLoad.material := '';
			loadStep := Surface.LEFT;
			RETURN;
		END_IF
		
		aoiLoad.surfaceID := Surface.BOTTOM;
		aoiLoad.material := pair.bottom;
		aoiLoad.suctions := suctionBottom;
		aoiLoad.numPads := UPPER_BOUND(suctionBottom, 1) - LOWER_BOUND(suctionBottom, 1) + 1;
		
		aoiLoad.execute := NOT aoiLoad.busy;
		
	Surface.LEFT:
		IF NOT includeLeft OR aoiLoad.donePulse THEN
			aoiLoad.execute := FALSE;
			aoiLoad.material := '';
			loadStep := Surface.RIGHT;
			RETURN;
		END_IF
		
		aoiLoad.surfaceID := Surface.LEFT;
		aoiLoad.material := pair.left;
		aoiLoad.suctions := suctionLeft;
		aoiLoad.numPads := UPPER_BOUND(suctionLeft, 1) - LOWER_BOUND(suctionLeft, 1) + 1;
		
		aoiLoad.execute := NOT aoiLoad.busy;
		
	Surface.RIGHT:
		IF NOT includeRight OR aoiLoad.donePulse THEN
			aoiLoad.execute := FALSE;
			aoiLoad.material := '';
			loadStep := COMPLETE;
			RETURN;
		END_IF
		
		aoiLoad.surfaceID := Surface.RIGHT;
		aoiLoad.material := pair.right;
		aoiLoad.suctions := suctionRight;
		aoiLoad.numPads := UPPER_BOUND(suctionRight, 1) - LOWER_BOUND(suctionRight, 1) + 1;
		
		aoiLoad.execute := NOT aoiLoad.busy;
		
	COMPLETE:				
		robot.release(sectionID);
		
		aoiLoad.material := '';
		aoiLoad.execute := FALSE;
		
		loadEx := TRUE;
END_CASE
END_METHOD

METHOD PROTECTED maintenance : BOOL
VAR_INPUT
END_VAR
{warning disable C0371}
//no specific tasks yet, free run and testing
SetSuctions(suctionTop, suctionEnableTop);
SetSuctions(suctionLeft, suctionEnableLeft);
SetSuctions(suctionRight, suctionEnableRight);
SetSuctions(suctionBottom, suctionEnableBottom);

IF robotLeft.Done THEN
	robotLeft.clearCommand();
END_IF

IF robotRight.Done THEN
	robotRight.clearCommand();
END_IF
END_METHOD

METHOD PROTECTED manual : BOOL
VAR_INPUT
END_VAR
END_METHOD

METHOD PROTECTED process : BOOL
VAR_INPUT
	auto : BOOL;
END_VAR
VAR_OUTPUT
	error : BOOL;
END_VAR
VAR
	currentPair : REFERENCE TO PositionMaterials REF= materialsArr[iPair];
END_VAR
{warning disable C0371}
IF iPair >= CONSTS.maxPairs THEN
	process := TRUE;
	RETURN;
ELSIF NOT PositionIsValid(pair := currentPair) THEN
	iPair := iPair + 1;
	RETURN;
END_IF

CASE step OF
	IDLE:
		IF auto OR_ELSE execute THEN
			step := STAGING;
		END_IF

	LOAD_WB:
		IF
			directionCheckAndSet(conveyorPos, currentPair.position) AND 
			( (auto AND done) OR_ELSE (NOT auto AND execute) )
		THEN
			robotLeft.clearCommand();
			robotRight.clearCommand();
			
			aoiLoadLeft.reset();
			aoiLoadRight.reset();
			
			loadStepLeft := loadStepRight := 0;
			stageStepLeft := stageStepRight := 0;
			
			done := FALSE;
			suctionEnableTop := suctionEnableLeft := suctionEnableRight := suctionEnableBottom := FALSE;
			execute := FALSE;
			
			step := PUSH;
			RETURN;
		END_IF
		
		IF NOT done THEN
			done := load(pairIndex := iPair, error => error);
		END_IF
		
		IF NOT auto THEN
			SetSuctions(suctionTop, suctionEnableTop);
			SetSuctions(suctionLeft, suctionEnableLeft);
			SetSuctions(suctionRight, suctionEnableRight);
			SetSuctions(suctionBottom, suctionEnableBottom);
		END_IF
		
	PUSH:
		IF
			(auto AND latchLeft AND latchRight AND pistonBottom.extended) OR_ELSE
			(NOT auto AND execute)
		THEN
			insertionLeft.stop();
			insertionRight.stop();
			
			latchLeft := latchRight := FALSE;
			execute := FALSE;
			step := STRAP;
			RETURN;
		END_IF
		
		IF NOT validateInsertion(checkTop:= FALSE, checkLeft:= FALSE, checkRight:= FALSE, checkBottom:= FALSE) THEN
			error := TRUE;
			RETURN;
		END_IF
		
		IF 
			insertionLeft.sliderPos <> demoHeight/2 OR 
			insertionRight.sliderPos <> demoHeight/2
		THEN
			insertionLeft.align(demoHeight/2);
			insertionRight.align(demoHeight/2);
			RETURN;
		END_IF
		
		
		IF insertionLeft.Contact THEN
			latchLeft := TRUE;
		ELSIF NOT latchLeft THEN
			insertionLeft.press();
		END_IF
		
		IF insertionRight.Contact THEN
			latchRight := TRUE;
		ELSIF NOT latchRight THEN
			insertionRight.press();
		END_IF
		pistonBottom.extend();
		
	STRAP:
		suctionRelease(IN:= , PT:= suctionReleaseDelay, Q=> , ET=> );
		
		strapper.bEnable := TRUE;
		IF strapper.done THEN
			suctionRelease.IN := FALSE;
			step := RELEASE;
			RETURN;
		END_IF
		
		IF suctionRelease.Q THEN
			SetSuctions(suctionTop, FALSE);
			SetSuctions(suctionLeft, FALSE);
			SetSuctions(suctionRight, FALSE);
			SetSuctions(suctionBottom, FALSE);
		ELSIF strapper.atBundleLevel THEN
			suctionRelease.IN := TRUE;
		END_IF
		
		IF strapper.ready THEN
			strapper.strap();
		END_IF
		
		IF execute THEN
			suctionRelease.IN := FALSE;
			execute := FALSE;
			step := RELEASE;
		END_IF
		
	RELEASE: //release command		
		insertionLeft.toHome();
		insertionRight.toHome();
		pistonBottom.retract();
		
		IF 
			(insertionLeft.screw.AtHome AND insertionRight.screw.AtHome AND pistonBottom.retracted) OR
			execute
		THEN
			execute := FALSE;
			step := COMPLETE;
		END_IF
	
	COMPLETE:
		//reset everything
		iPair := iPair + 1;
		step := IDLE;
END_CASE
END_METHOD

METHOD PROTECTED ps_AbortCondition : BOOL
VAR_INPUT
END_VAR
{warning disable C0371}
ps_AbortCondition :=
	insertionLeft.error OR 
	insertionRight.error OR 
	robotLeft.error OR 
	robotRight.error OR
	strapper.error;
END_METHOD

METHOD PROTECTED ps_Aborted : BOOL
VAR_INPUT
END_VAR
ps_Aborted := TRUE;
END_METHOD

METHOD PROTECTED ps_Aborting : BOOL
VAR_INPUT
END_VAR
{warning disable C0371}
insertionLeft.stop();
insertionRight.stop();
pistonBottom.stop();

aoiLoadLeft.reset();
aoiLoadRight.reset();

aoiStageLeft.reset();
aoiStageRight.reset();

robotLeft.clearCommand();
robotRight.clearCommand();

//stop conveyors

ps_Aborting :=
	NOT insertionLeft.active AND
	NOT insertionRight.active AND
	NOT pistonBottom.busy AND
	NOT robotLeft.Busy AND
	NOT robotRight.Busy;
END_METHOD

METHOD PROTECTED ps_Clearing : BOOL
VAR_INPUT
END_VAR
{warning disable C0371}
insertionLeft.reset();
insertionRight.reset();

ps_Clearing := 
	NOT insertionLeft.error AND
	NOT insertionRight.error AND
	NOT strapper.error AND
	NOT robotLeft.error AND
	NOT robotRight.error;
END_METHOD

METHOD PROTECTED ps_Complete : BOOL
VAR_INPUT
END_VAR
ps_Complete := TRUE;
END_METHOD

METHOD PROTECTED ps_Completing : BOOL
VAR_INPUT
END_VAR
ps_Completing := NOT occupied;
END_METHOD

METHOD PROTECTED ps_Execute : BOOL
VAR_INPUT
END_VAR
VAR_OUTPUT
	error : BOOL;
END_VAR
SUPER^.ps_Execute();
END_METHOD

METHOD PROTECTED ps_Held : BOOL
VAR_INPUT
END_VAR
ps_Held := NOT hold;
END_METHOD

METHOD PROTECTED ps_HoldCondition : BOOL
VAR_INPUT
END_VAR
END_METHOD

METHOD PROTECTED ps_Holding : BOOL
VAR_INPUT
END_VAR
{warning disable C0371}
insertionLeft.stop();
insertionRight.stop();
pistonBottom.stop();
//set robot to pause

ps_Holding :=
	NOT insertionLeft.active AND
	NOT insertionRight.active;
END_METHOD

METHOD PROTECTED ps_Idle : BOOL
VAR_INPUT
END_VAR
ps_Idle := execute;
execute := FALSE;
END_METHOD

METHOD PROTECTED ps_Resetting : BOOL
VAR_INPUT
END_VAR
{warning disable C0371}
insertionLeft.reset();
insertionRight.reset();

ps_Resetting := 
	reset AND
	NOT insertionLeft.error AND
	NOT insertionRight.error AND
	NOT strapper.error AND
	NOT robotLeft.error AND
	NOT robotRight.error;
END_METHOD

METHOD PROTECTED ps_Starting : BOOL
VAR_INPUT
END_VAR
{warning disable C0371}
robotLeft.clearCommand();
robotRight.clearCommand();

insertionLeft.homingSequence();
insertionRight.homingSequence();
pistonBottom.retract();

ps_Starting := 
	insertionLeft.screw.HomeSet AND 
	insertionRight.screw.HomeSet AND 
	pistonBottom.retracted;
END_METHOD

METHOD PROTECTED ps_StopCondition : BOOL
VAR_INPUT
END_VAR
ps_StopCondition := 
	stop;
END_METHOD

METHOD PROTECTED ps_Stopped : BOOL
VAR_INPUT
END_VAR
ps_Stopped := TRUE;
END_METHOD

METHOD PROTECTED ps_Stopping : BOOL
VAR_INPUT
END_VAR
{warning disable C0371}
insertionLeft.stop();
insertionRight.stop();
pistonBottom.stop();

aoiLoadLeft.reset();
aoiLoadRight.reset();

aoiStageLeft.reset();
aoiStageRight.reset();

robotLeft.clearCommand();
robotRight.clearCommand();

//stop conveyors

ps_Stopping :=
	NOT insertionLeft.active AND
	NOT insertionRight.active AND
	NOT pistonBottom.busy AND
	NOT robotLeft.Busy AND
	NOT robotRight.Busy;
END_METHOD

METHOD PROTECTED ps_SuspendCondition : BOOL
VAR_INPUT
END_VAR
END_METHOD

METHOD PROTECTED ps_Suspended : BOOL
VAR_INPUT
END_VAR
ps_Suspended := NOT ps_SuspendCondition();
END_METHOD

METHOD PROTECTED ps_Suspending : BOOL
VAR_INPUT
END_VAR
ps_Suspending := TRUE;
END_METHOD

METHOD PROTECTED ps_Unholding : BOOL
VAR_INPUT
END_VAR
ps_Unholding := TRUE;
END_METHOD

METHOD PROTECTED ps_Unsuspending : BOOL
VAR_INPUT
END_VAR
ps_Unsuspending := TRUE;
END_METHOD

METHOD PROTECTED FINAL runSectionTasks : BOOL
VAR_INPUT
	auto : BOOL;
END_VAR
VAR_OUTPUT
	error : BOOL;
END_VAR
SUPER^.runSectionTasks(auto := auto, error => error);

CASE status OF //add additional instructions for each state
	SectionTask.IDLE:
		//
	
	SectionTask.ALIGNING:
		stage(error => error);
		
	SectionTask.ACTIVE:
		//
		
	SectionTask.CLEARING:
		aoiLoadLeft.reset();
		aoiLoadRight.reset();
		
		aoiStageLeft.reset();
		aoiStageRight.reset();
		
		aoiTemplateLeft.reset();
		aoiTemplateRight.reset();
		
	SectionTask.COMPLETE:	
		//
		
	-100:
		//
		
END_CASE
END_METHOD

METHOD PROTECTED stage : BOOL
VAR_OUTPUT
	error : BOOL;
END_VAR
{warning disable C0371}

(*
this method only exists to call stageEx() for both robots
*)
(*
stage := leftDone AND rightDone;

IF NOT leftDone THEN
	leftDone := stageEx(
		robot:= robotLeft, 
		aoiTemplate:= aoiTemplateLeft, 
		aoiStaging:= aoiStageLeft, 
		stageStep:= stageStepLeft, 
		//iSlot:= iSlotLeft, 
		includeTop:= TRUE, 
		includeLeft:= TRUE, 
		includeRight:= FALSE, 
		includeBottom:= FALSE, 
		error=> );
END_IF

IF NOT rightDone THEN
	rightDone := stageEx(
		robot:= robotRight, 
		aoiTemplate:= aoiTemplateRight, 
		aoiStaging:= aoiStageRight, 
		stageStep:= stageStepRight, 
		//iSlot:= iSlotRight, 
		includeTop:= FALSE, 
		includeLeft:= FALSE, 
		includeRight:= TRUE, 
		includeBottom:= TRUE, 
		error=> );
END_IF
*)

stage := 
	stageEx(
		robot:= robotLeft, 
		aoiTemplate:= aoiTemplateLeft, 
		aoiStaging:= aoiStageLeft, 
		stageStep:= stageStepLeft, 
		includeTop:= TRUE, 
		includeLeft:= TRUE, 
		includeRight:= FALSE, 
		includeBottom:= FALSE, 
		error=> )
	AND
	stageEx(
		robot:= robotRight, 
		aoiTemplate:= aoiTemplateRight, 
		aoiStaging:= aoiStageRight, 
		stageStep:= stageStepRight, 
		includeTop:= FALSE, 
		includeLeft:= FALSE, 
		includeRight:= TRUE, 
		includeBottom:= TRUE, 
		error=> );
END_METHOD

METHOD PRIVATE stageEx : BOOL
VAR_IN_OUT
	robot : RobotA21;
	aoiTemplate : AOI_StagingTemplate;
	aoiStaging : AOI_StageWoodBunk;
	stageStep : INT;
END_VAR
VAR_INPUT
	includeTop, includeLeft, includeRight, includeBottom : BOOL;
END_VAR
VAR_OUTPUT
	error : BOOL;
END_VAR
{warning disable C0371}
IF robot.error THEN
	error := TRUE;
	RETURN;
ELSIF robot.reservation <> sectionID AND_THEN NOT robot.reserve(sectionID) THEN
	RETURN;
ELSIF robot.tool <> sectionID AND_THEN NOT robot.changeEOAT(targetTool := sectionID) THEN
	RETURN;
END_IF

CASE stageStep OF
	0: //generate staging template
		IF aoiTemplate.done THEN
			aoiTemplate.execute := FALSE;
			stageStep := 10;
			RETURN;
		END_IF
		
		aoiTemplate.execute := NOT aoiTemplate.busy;
		
		aoiTemplate.includeTop := includeTop;
		aoiTemplate.includeLeft := includeLeft;
		aoiTemplate.includeRight := includeRight;
		aoiTemplate.includeBottom := includeBottom;
		
	10: //stage tables
		IF aoiStaging.slot > 10 THEN
			aoiStaging.execute := FALSE;			
			stageStep := COMPLETE;
			RETURN;
		END_IF
		
		aoiStaging.execute := NOT aoiStaging.busy; //execute if aoiStaging is ready
		
		aoiStaging.slot := MAX(1, aoiStaging.slot); //if 0, sets to 1
		aoiStaging.slot := MIN(aoiStaging.slot, 999); //prevents overflow 
		
		IF aoiStaging.donePulse THEN
			aoiStaging.slot := aoiStaging.slot + 1;
		END_IF
	
	COMPLETE:
		aoiTemplate.clearTemplate();
		aoiTemplate.execute := FALSE;
		aoiStaging.execute := FALSE;
		aoiStaging.reset();
		
		robot.release(sectionID);
		
		aoiStaging.slot := 0;
		
		stageEx := TRUE;
		//stageStep := 0;
END_CASE

error := aoiStaging.error;
END_METHOD

METHOD PROTECTED unload : BOOL
VAR_INPUT
END_VAR
//unload from insertion
//remove from staging table
END_METHOD

METHOD PROTECTED validateInsertion : BOOL
VAR_INPUT
	checkTop : BOOL;
	checkLeft : BOOL;
	checkRight : BOOL;
	checkBottom : BOOL;
END_VAR
validateInsertion := 
	(NOT checkTop OR_ELSE SuctionQuality(suctions:= suctionTop)) AND
	(NOT checkLeft OR_ELSE SuctionQuality(suctions:= suctionLeft)) AND
	(NOT checkRight OR_ELSE SuctionQuality(suctions:= suctionRight)) AND
	(NOT checkBottom OR_ELSE SuctionQuality(suctions:= suctionBottom));

(*
validateSuctionQuality := 
	(
		NOT checkTop OR_ELSE InsertionQuality(
			suctions:= suctionTop, 
			insertionMaterial:= loadedMaterials[Surface.TOP], 
			recipeMaterial:= materialsArr[iPair].top)
	) AND
	(
		NOT checkLeft OR_ELSE InsertionQuality(
			suctions:= suctionLeft, 
			insertionMaterial:= loadedMaterials[Surface.LEFT], 
			recipeMaterial:= materialsArr[iPair].left)
	) AND
	(
		NOT checkRight OR_ELSE InsertionQuality(
			suctions:= suctionRight, 
			insertionMaterial:= loadedMaterials[Surface.RIGHT], 
			recipeMaterial:= materialsArr[iPair].right)
	) AND
	(
		NOT checkBottom OR_ELSE InsertionQuality(
			suctions:= suctionBottom, 
			insertionMaterial:= loadedMaterials[Surface.BOTTOM], 
			recipeMaterial:= materialsArr[iPair].bottom)
	);
*)
END_METHOD

END_FUNCTION_BLOCK

// ---- Sections/A21b - Wood Bunk/AOIs/AOI_StagingTemplate.TcPOU
FUNCTION_BLOCK AOI_StagingTemplate
VAR_INPUT
	execute : BOOL;
END_VAR
VAR_IN_OUT
	materialsArr : ARRAY[*] OF PositionMaterials; //[0..GVL.maxPairs]
	table : StagingTable;
END_VAR
VAR_INPUT
	includeTop, includeLeft, includeRight, includeBottom : BOOL; 
END_VAR
VAR_OUTPUT
	busy : BOOL;
	done : BOOL;
END_VAR
VAR
	trigger : R_TRIG;
	run : BOOL;
	step : (IDLE, GENERATE, COMPLETE);
	i : INT;
END_VAR
VAR	
	stagingArray : ARRAY[0..(Consts.maxPairs+1)*2] OF STRING;
	
	template : StagingTable;
	templateSlots AT %M* : ARRAY[1..10] OF MaterialSlot;
END_VAR

{warning disable C0371}

template(slots:= templateSlots);

trigger(CLK:= execute, Q=> run);

CASE step OF
	IDLE:
		IF run THEN
			step := GENERATE;
			done := FALSE;
		END_IF
		
	GENERATE:
		//strings contain garbage chars after a null byte, they must be manually cleaned before checking if they are byte-empty
		CleanStringsArray(arr := stagingArray);
		IF DataIsEmpty(arr := ADR(stagingArray), arrSize := SIZEOF(stagingArray)) THEN //if staging array is empty, fill the array
			createStagingArray(
				includeTop:= includeTop, 
				includeLeft:= includeLeft, 
				includeRight:= includeRight, 
				includeBottom:= includeBottom);
		END_IF
		
		//copy over the real slots before autofilling, otherwise the template may fill occupied slots
		table.copyFrom(src := table);
		
		(*
		iterate through all pairs and autofill the template
		replace succesfully autofilled materials with empty string
		if staging needs to be performed a 2nd time, autofilling empty strings is always unsuccessful
		*)
		FOR i:=0 TO (CONSTS.maxPairs+1)*2 BY 1 DO
			IF template.autofill(material := stagingArray[i]) THEN
				stagingArray[i] := '';
			END_IF
		END_FOR
		
		step := COMPLETE;
	
	COMPLETE:
		done := TRUE;
		
		step := IDLE;
		
END_CASE

busy := run OR step > 0;

METHOD PRIVATE addToStagingArray : BOOL
VAR_INPUT
	material : STRING;
END_VAR
VAR
	remainingMaterial : STRING;
	splitMaterial : STRING;
END_VAR
remainingMaterial := material;
WHILE FIND(remainingMaterial, '_') > 0 DO
	splitCombinedMaterials(remainingMaterial, splitMaterial);
	IF splitMaterial <> '' THEN
		AddToStringArray(arr := stagingArray, newString := splitMaterial, numElements => , nextIndex => );
	END_IF
END_WHILE

IF remainingMaterial <> '' THEN
	AddToStringArray(arr := stagingArray, newString := remainingMaterial, numElements => , nextIndex => );
END_IF

addToStagingArray := TRUE;
END_METHOD

METHOD clearArray : BOOL
VAR_INPUT
END_VAR
MEMSET(ADR(stagingArray), 0, SIZEOF(stagingArray));
END_METHOD

METHOD clearTemplate : BOOL
VAR_INPUT
END_VAR
template.clear();
END_METHOD

METHOD PRIVATE createStagingArray : BOOL
VAR_INPUT
	includeTop : BOOL;
	includeLeft : BOOL;
	includeRight : BOOL;
	includeBottom : BOOL;
END_VAR
VAR
	remainingMaterial : STRING;
	splitMaterial : STRING;
	
	i : INT;
END_VAR
FOR i:=0 TO CONSTS.maxPairs BY 1 DO
	IF includeTop THEN
		addToStagingArray(material := materialsArr[i].top);
	END_IF
	
	IF includeLeft THEN
		addToStagingArray(material := materialsArr[i].left);
	END_IF
	
	IF includeRight THEN
		addToStagingArray(material := materialsArr[i].right);
	END_IF
	
	IF includeBottom THEN
		addToStagingArray(material := materialsArr[i].bottom);
	END_IF
END_FOR
END_METHOD

METHOD getSlot : STRING
VAR_INPUT
	i : INT;
END_VAR
VAR_OUTPUT
	error : BOOL;
END_VAR
getSlot := template.getSlot(i := i, error => error);
END_METHOD

METHOD reset : BOOL
VAR_INPUT
END_VAR
VAR
	temp : AOI_StagingTemplate;
END_VAR
//(*
busy := FALSE;
done := FALSE;
step := 0;

clearArray();
clearTemplate();
//*)
//THIS^ := temp;
END_METHOD

METHOD PRIVATE splitCombinedMaterials : BOOL
VAR_IN_OUT
	materialID : STRING;
	splitMaterial : STRING;
END_VAR
VAR
	i : INT;
END_VAR
FindAndSplitChar(
	sSeparatorChar:= '_', 
	pSrcString:= ADR(materialID), 
	
	pLeftString:= ADR(splitMaterial), 
	nLeftSize:= SIZEOF(splitMaterial), 
	
	pRightString:= ADR(materialID), 
	nRightSize:= SIZEOF(materialID), 
	
	bSearchFromRight:= FALSE);
END_METHOD

END_FUNCTION_BLOCK

// ---- Sections/A21b - Wood Bunk/AOIs/AOI_LoadWoodBunk.TcPOU
FUNCTION_BLOCK AOI_LoadWoodBunk
VAR_INPUT
	execute : BOOL;
END_VAR
VAR_IN_OUT CONSTANT
	sectionID : SectionEnum;
END_VAR
VAR_IN_OUT
	robot : RobotA21;
	table : StagingTable;
	suctions : ARRAY[*] OF SuctionPad;
	//if assigned using . operator instead of (), this becomes a pointer - use numPads isntead of UPPER_BOUND/LOWER_BOUND
	loadedMaterials : ARRAY[*] OF STRING;
END_VAR
VAR_INPUT
	surfaceID : Surface;
	material : STRING;	
	numPads : DINT;
END_VAR
VAR_OUTPUT
	busy : BOOL;
	done : BOOL;
	error : BOOL;
	
	recovery : BOOL;
	failCounter : INT;
	
	donePulse : BOOL;
END_VAR
VAR
	run : BOOL;
	trigger : R_TRIG;
	doneTrigger : R_TRIG;
	
	slot : INT;
	
	suctionTimer : TON;
	step : (IDLE, PREP_ROBOT, GET_FROM_TABLE, LOAD_TO_INSERTION, COMPLETE, RECOVERY_IDLE, RECOVERY_REMOVE, RECOVERY_STAGE);
END_VAR
VAR
	i : DINT;
	test : BOOL;
END_VAR
VAR CONSTANT
	suctionDelay : TIME := T#2S;
	suctionDistance : INT := 10;
END_VAR

{warning disable C0371}

trigger(CLK:= execute, Q=> );
doneTrigger(CLK:= done, Q=> donePulse);
busy := trigger.Q OR step > 0;

IF step > IDLE AND_THEN NOT preExecution() THEN //conditions to track before execution
	RETURN;
END_IF

(*
if required bunk was not found on table - restage entire table
if bunk was not loaded correctly - remove bunk, then restage entire table
*)

CASE step OF
	IDLE:
		IF trigger.Q THEN //reset outputs
			done := FALSE;
			error := FALSE;
			recovery := FALSE;
			
			step := PREP_ROBOT;
		END_IF
		
	PREP_ROBOT:
		robot.clearCommand();
		IF robot.Ready THEN
			step := GET_FROM_TABLE;
			slot := 0;
		END_IF
		
	GET_FROM_TABLE:		
		IF slot < 1 AND_THEN NOT table.findSlot(material := material, index => slot) THEN
			step := RECOVERY_STAGE;
			RETURN;
		END_IF
		
		IF NOT table.isOccupied(i := slot) AND table.getSlot(i := slot) <> '' THEN //move from table to robot gripper
			robot.HoldMaterial := table.getSlot(i := slot);
			table.remove(i := slot, material => );
		END_IF
		
		IF robot.Done THEN
			step := COMPLETE;
			RETURN;
		ELSIF robot.materialAtHoldingPosition >= 1 AND robot.materialAtHoldingPosition <= 8 THEN
			step := LOAD_TO_INSERTION;
			RETURN;
		END_IF
		
		CASE surfaceID OF
			Surface.TOP: 					robot.setGroup(group := 1, value := TaskA21.LOAD_BUNK_TOP); 
			Surface.LEFT, Surface.RIGHT: 	robot.setGroup(group := 1, value := TaskA21.LOAD_BUNK_SIDE);
			Surface.BOTTOM: 				robot.setGroup(group := 1, value := TaskA21.LOAD_BUNK_BOTTOM);
		END_CASE
		robot.setGroup(group := 2, value := slot); 
			
	LOAD_TO_INSERTION:
		IF robot.materialAtHoldingPosition > 0 AND robot.HoldMaterial <> '' THEN //move from gripper to insertion
			IF loadedMaterials[surfaceID] = '' THEN //transfer to insertion as is
				loadedMaterials[surfaceID] := robot.HoldMaterial;
			ELSE //join with existing material using underscore _
				loadedMaterials[surfaceID] := JoinStrings(loadedMaterials[surfaceID], robot.HoldMaterial, '_');
			END_IF
			robot.HoldMaterial := '';
		END_IF
		
		CASE surfaceID OF
			Surface.TOP, Surface.BOTTOM:	SetSuctionsPtr(suctions := suctions, numPads := numPads, state := TRUE);
			Surface.LEFT, Surface.RIGHT:	SetSuctionsPtr(suctions := suctions, numPads := numPads, state := TRUE);
		END_CASE
		
		IF robot.Done THEN
			suctionTimer.IN := FALSE;
			step := COMPLETE;
			RETURN;
		END_IF
		
		suctionTimer(IN:= , PT:= suctionDelay, Q=> , ET=> );
		suctionTimer.IN := TRUE;
		
		IF suctionTimer.Q THEN
			robot.setGroup(group := 9, value := robot.materialAtHoldingPosition);
		END_IF
	
	COMPLETE:
		robot.clearCommand();
		
		//check insertion quality
		IF InsertionQuality(suctions := suctions, insertionMaterial := loadedMaterials[surfaceID], recipeMaterial := material) THEN
			done := TRUE;
			slot := 0;
			step := 0;
		ELSE //recovery - restage table
			failCounter := failCounter + 1;
			step := RECOVERY_IDLE;
		END_IF
		
	//---------RECOVERY-----------------------------------------
	RECOVERY_IDLE:
		robot.clearCommand();
		IF robot.Ready THEN
			step := RECOVERY_REMOVE;
		END_IF
		
	RECOVERY_REMOVE:
		IF robot.Done THEN
			step := RECOVERY_STAGE;
			RETURN;
		END_IF
		
		CASE surfaceID OF
			Surface.TOP:					robot.setGroup(group := 1, value := TaskA21.REMOVE_BUNK_TOP);
			Surface.LEFT, Surface.RIGHT:	robot.setGroup(group := 1, value := TaskA21.REMOVE_BUNK_SIDE);
			Surface.BOTTOM:					robot.setGroup(group := 1, value := TaskA21.REMOVE_BUNK_BOTTOM);
		END_CASE
	
	RECOVERY_STAGE:	
		recovery := TRUE;
		error := TRUE;
		
END_CASE

METHOD PRIVATE preExecution : BOOL
VAR_INPUT
END_VAR
{warning disable C0371}
IF material = '' THEN
	done := TRUE;
	RETURN;
END_IF

IF //robot must be ready before execution
	robot.error OR 
	robot.reservation <> sectionID OR 
	robot.tool <> sectionID
THEN
	error := TRUE;
	RETURN;
END_IF

preExecution := TRUE;
END_METHOD

METHOD reset : BOOL
VAR_INPUT
END_VAR
VAR
	temp : AOI_LoadWoodBunk;
END_VAR
//(*
done := FALSE;
error := FALSE;
recovery := FALSE;
slot := 0;
step := 0;

failCounter := 0;
//*)
//THIS^ := temp;
END_METHOD

END_FUNCTION_BLOCK

// ---- HARDWARE_DISTRUBUTION/A26.TcPOU
PROGRAM A26
VAR_IN_OUT
	spacerRecollector : SpacerRecollectionUnit;
END_VAR
VAR
	robot7 : RobotA26; //placeholder, will need another robot definition for A26
	robotSliderA26 : ServoNC;
END_VAR
VAR //sensors to detect spacer on transfer conveyors
	spacerPresent_A24_LRC_C02 AT %I* : BOOL;
	spacerPresent_A24_LRC_C04 AT %I* : BOOL;
	spacerPresent_A24_LRC_C06 AT %I* : BOOL;
	spacerPresent_A24_LRC_C08 AT %I* : BOOL;
	spacerPresent_A24_LRC_C10 AT %I* : BOOL;
	spacerPresent_A24_LRC_C12 AT %I* : BOOL;
END_VAR

callHardware();
setupHardware();
runModules();
callHardware();

METHOD PRIVATE callHardware : BOOL
VAR_INPUT
END_VAR
robot7();	
robotSliderA26(bEnable:= TRUE, ready=> , position=> , velocity=> );
END_METHOD

METHOD PRIVATE runModules : BOOL
VAR_INPUT
END_VAR
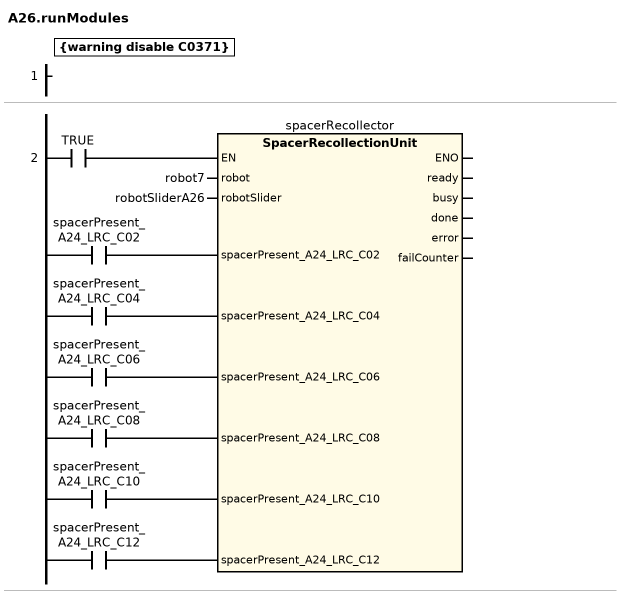
// NETWORK 1
// label: {warning disable C0371}

// NETWORK 2
spacerRecollector(
    robot := robot7,
    robotSlider := robotSliderA26,
    spacerPresent_A24_LRC_C02 := spacerPresent_A24_LRC_C02,
    spacerPresent_A24_LRC_C04 := spacerPresent_A24_LRC_C04,
    spacerPresent_A24_LRC_C06 := spacerPresent_A24_LRC_C06,
    spacerPresent_A24_LRC_C08 := spacerPresent_A24_LRC_C08,
    spacerPresent_A24_LRC_C10 := spacerPresent_A24_LRC_C10,
    spacerPresent_A24_LRC_C12 := spacerPresent_A24_LRC_C12); // SpacerRecollectionUnit
END_METHOD

METHOD PRIVATE setupHardware : BOOL
VAR
	iCornerGuardSlot : CornerGuard;
	iCardboardSlot : Cardboard;
	i : INT;
END_VAR
END_METHOD

END_PROGRAM

// ---- HARDWARE_DISTRUBUTION/A22.TcPOU
PROGRAM A22
VAR_IN_OUT
	sectionCC : CardboardEx;
	
	bundlesQueue : ARRAY[0..CONSTS.maxQueue] OF Bundle;
	bundlesBypass : ARRAY[0..CONSTS.maxQueue] OF BOOL;
END_VAR
VAR_OUTPUT //conveyors only
	A22_SC_C15 		: ConveyorSC;
	A22_LSC_C16 	: ConveyorLSC;
	A22_LSC_C17 	: ConveyorLSC;
END_VAR
VAR
	robot3, robot4 : RobotA22;
	
	benderA22Left : FoldingMachine;
	
	skidA22Left, skidA22Right : SkidMagazine;
	magazineA22Left, magazineA22Right : SkidMagazine;
	
	wrapperA22 : WrapMachine;
	overhead : STRING;
	
	horizontalDriveA22Left, horizontalDriveA22Right : ServoNC := (
		limitSensorDefaultState := TRUE);
		
	verticalDriveA22Left, verticalDriveA22Right : ClearLinkMC := (
		limitSensorDefaultState := TRUE, 
		homingDirectionOut := TRUE, //outwards (up)
		minPosition := (26*5 * 25.4),
		displacementPerRotation := 5,
		unitsPerPulse := 800); //800 counts = 1 rotation
		
	insertionA22Left, insertionA22Right : Insertion;

	pistonA22Bottom : SimplePiston;
	
	(*
	each insertion suction array has 3 pads
	[1] - top/bottom
	[2] - corner
	[3] - side
	*)
	suctionA22TopLeft : ARRAY[1..3] OF SuctionPad;
	suctionA22TopRight : ARRAY[1..3] OF SuctionPad;
	suctionA22BottomLeft : ARRAY[1..3] OF SuctionPad; 
	suctionA22BottomRight : ARRAY[1..3] OF SuctionPad;
	
	suctionA22Bottom : ARRAY[1..2] OF SuctionPad;
END_VAR
VAR //data arrays to be passed into material holder FBs - do not access directly
	skidHmiA22Left, skidHmiA22Right AT %M* : ARRAY[1...Cardboard.size-1] OF MaterialSlot;
	magazineHmiA22Left, magazineHmiA22Right AT %M* : ARRAY[1..CornerGuard.size-1] OF MaterialSlot;
END_VAR
VAR //other
	conveyorsCC : ARRAY[1..3] OF POINTER TO ConveyorSC;
END_VAR

callHardware();

setupHardware();

runModules();

callHardware();

METHOD PRIVATE callHardware : BOOL
skidA22Left(slots := skidHmiA22Left);
skidA22Right(slots := skidHmiA22Right);
magazineA22Left(slots := magazineHmiA22Left);
magazineA22Right(slots := magazineHmiA22Right);

wrapperA22(extSafety := robot3.wrapSafetyIn AND robot4.wrapSafetyIn);

verticalDriveA22Left(
	bEnable:= , 
	pulse=> , 
	brakeRelease=> , 
	enable=> , 
	A=> , 
	B=> , 
	clear=> );
verticalDriveA22Right(
	bEnable:= , 
	pulse=> , 
	brakeRelease=> , 
	enable=> , 
	A=> , 
	B=> , 
	clear=> );

horizontalDriveA22Left(bEnable:= TRUE, ready=> , position=> , velocity=> );
horizontalDriveA22Right(bEnable:= TRUE, ready=> , position=> , velocity=> );

insertionA22Left(
	slider:= verticalDriveA22Left, 
	screw:= horizontalDriveA22Left, 
	contact=> , 
	active=> , 
	error=> , 
	home=> , 
	homingComplete=> , 
	sliderPos=> );
	
insertionA22Right(
	slider:= verticalDriveA22Right, 
	screw:= horizontalDriveA22Right, 
	contact=> , 
	active=> , 
	error=> , 
	home=> , 
	homingComplete=> , 
	sliderPos=> );
END_METHOD

METHOD PRIVATE runModules : BOOL
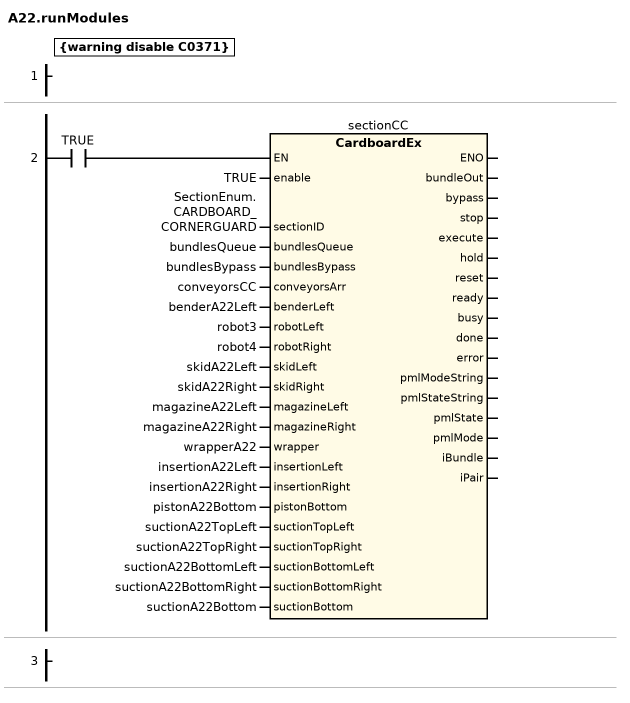
// NETWORK 1
// label: {warning disable C0371}

// NETWORK 2
sectionCC(
    enable := TRUE,
    sectionID := SectionEnum.CARDBOARD_CORNERGUARD,
    bundlesQueue := bundlesQueue,
    bundlesBypass := bundlesBypass,
    conveyorsArr := conveyorsCC,
    benderLeft := benderA22Left,
    robotLeft := robot3,
    robotRight := robot4,
    skidLeft := skidA22Left,
    skidRight := skidA22Right,
    magazineLeft := magazineA22Left,
    magazineRight := magazineA22Right,
    wrapper := wrapperA22,
    insertionLeft := insertionA22Left,
    insertionRight := insertionA22Right,
    pistonBottom := pistonA22Bottom,
    suctionTopLeft := suctionA22TopLeft,
    suctionTopRight := suctionA22TopRight,
    suctionBottomLeft := suctionA22BottomLeft,
    suctionBottomRight := suctionA22BottomRight,
    suctionBottom := suctionA22Bottom); // CardboardEx

// NETWORK 3
END_METHOD

